LIN {X 0,Y 291.883,Z 681.921,A -85,B 0,C 180,E1 -16741.379,E2 -16741.379} C_VEL
LIN {X 0,Y 291.735,Z 681.939,A -85,B 0,C 180,E1 -16746.918,E2 -16746.918} C_VEL
LIN {X 0,Y 291.622,Z 681.967,A -85,B 0,C 180,E1 -16749.712,E2 -16749.712} C_VEL
LIN {X 0,Y 291.513,Z 681.968,A -85,B 0,C 180,E1 -16753.95,E2 -16753.95} C_VEL
LIN {X 0,Y 291.479,Z 681.972,A -85,B 0,C 180,E1 -16756.818,E2 -16756.818} C_VEL
LIN {X 0,Y 291.477,Z 681.99,A -85,B 0,C 180,E1 -16759.893,E2 -16759.893} C_VEL
LIN {X 0,Y 291.416,Z 681.996,A -85,B 0,C 180,E1 -16764.203,E2 -16764.203} C_VEL
LIN {X 0,Y 291.414,Z 681.938,A -85,B 0,C 180,E1 -16767.272,E2 -16767.272} C_VEL
LIN {X 0,Y 291.329,Z 681.954,A -85,B 0,C 180,E1 -16770.437,E2 -16770.437} C_VEL
LIN {X 0,Y 291.337,Z 681.982,A -85,B 0,C 180,E1 -16773.699,E2 -16773.699} C_VEL
LIN {X 0,Y 291.422,Z 682.063,A -85,B 0,C 180,E1 -16777.556,E2 -16777.556} C_VEL
LIN {X 0,Y 291.562,Z 682.874,A -85,B 0,C 180,E1 -16777.957,E2 -16777.957} C_VEL
LIN {X 0,Y 292.964,Z 685.685,A -85,B 0,C 180,E1 -16778.482,E2 -16778.482} C_VEL
LIN {X 0,Y 295.139,Z 687.721,A -85,B 0,C 180,E1 -16779.091,E2 -16779.091} C_VEL
LIN {X 0,Y 297.372,Z 691.036,A -85,B 0,C 180,E1 -16779.745,E2 -16779.745} C_VEL
LIN {X 0,Y 299.349,Z 693.065,A -85,B 0,C 180,E1 -16780.308,E2 -16780.308} C_VEL
LIN {X 0,Y 302.176,Z 696.689,A -85,B 0,C 180,E1 -16781.129,E2 -16781.129} C_VEL
LIN {X 0,Y 304.398,Z 698.863,A -85,B 0,C 180,E1 -16781.754,E2 -16781.754} C_VEL
LIN {X 0,Y 307.399,Z 702.53,A -85,B 0,C 180,E1 -16782.702,E2 -16782.702} C_VEL
LIN {X 0,Y 309.651,Z 704.604,A -85,B 0,C 180,E1 -16783.366,E2 -16783.366} C_VEL
LIN {X 0,Y 312.93,Z 708.385,A -85,B 0,C 180,E1 -16784.462,E2 -16784.462} C_VEL
LIN {X 0,Y 315.506,Z 710.671,A -85,B 0,C 180,E1 -16785.293,E2 -16785.293} C_VEL
LIN {X 0,Y 318.764,Z 714.434,A -85,B 0,C 180,E1 -16786.475,E2 -16786.475} C_VEL
LIN {X 0,Y 321.428,Z 716.849,A -85,B 0,C 180,E1 -16787.424,E2 -16787.424} C_VEL
LIN {X 0,Y 324.974,Z 720.767,A -85,B 0,C 180,E1 -16788.792,E2 -16788.792} C_VEL
LIN {X 0,Y 327.213,Z 722.862,A -85,B 0,C 180,E1 -16789.66,E2 -16789.66} C_VEL
LIN {X 0,Y 330.789,Z 726.747,A -85,B 0,C 180,E1 -16791.088,E2 -16791.088} C_VEL
LIN {X 0,Y 333.202,Z 728.975,A -85,B 0,C 180,E1 -16792.056,E2 -16792.056} C_VEL
LIN {X 0,Y 336.504,Z 732.572,A -85,B 0,C 180,E1 -16793.429,E2 -16793.429} C_VEL
LIN {X 0,Y 339.383,Z 735.138,A -85,B 0,C 180,E1 -16794.624,E2 -16794.624} C_VEL
LIN {X 0,Y 343.284,Z 739.204,A -85,B 0,C 180,E1 -16796.335,E2 -16796.335} C_VEL
LIN {X 0,Y 346.175,Z 741.646,A -85,B 0,C 180,E1 -16797.613,E2 -16797.613} C_VEL
LIN {X 0,Y 349.884,Z 745.493,A -85,B 0,C 180,E1 -16799.349,E2 -16799.349} C_VEL
LIN {X 0,Y 352.817,Z 747.883,A -85,B 0,C 180,E1 -16800.742,E2 -16800.742} C_VEL
LIN {X 0,Y 356.182,Z 751.516,A -85,B 0,C 180,E1 -16802.455,E2 -16802.455} C_VEL
LIN {X 0,Y 359.846,Z 754.425,A -85,B 0,C 180,E1 -16804.388,E2 -16804.388} C_VEL
LIN {X 0,Y 363.148,Z 758.001,A -85,B 0,C 180,E1 -16806.288,E2 -16806.288} C_VEL
LIN {X 0,Y 366.688,Z 760.486,A -85,B 0,C 180,E1 -16808.414,E2 -16808.414} C_VEL
LIN {X 0,Y 367.985,Z 761.786,A -85,B 0,C 180,E1 -16809.246,E2 -16809.246} C_VEL
LIN {X 0,Y 370.733,Z 764.739,A -85,B 0,C 180,E1 -16811.2,E2 -16811.2} C_VEL
LIN {X 0,Y 373.538,Z 766.766,A -85,B 0,C 180,E1 -16813.28,E2 -16813.28} C_VEL
LIN {X 0,Y 375.474,Z 767.943,A -85,B 0,C 180,E1 -16814.874,E2 -16814.874} C_VEL
LIN {X 0,Y 377.522,Z 770.55,A -85,B 0,C 180,E1 -16816.885,E2 -16816.885} C_VEL
LIN {X 0,Y 379.42,Z 772.303,A -85,B 0,C 180,E1 -16819.024,E2 -16819.024} C_VEL
LIN {X 0,Y 381.332,Z 773.414,A -85,B 0,C 180,E1 -16821.522,E2 -16821.522} C_VEL
LIN {X 0,Y 382.798,Z 774.146,A -85,B 0,C 180,E1 -16824.133,E2 -16824.133} C_VEL
LIN {X 0,Y 383.462,Z 774.602,A -85,B 0,C 180,E1 -16825.796,E2 -16825.796} C_VEL
LIN {X 0,Y 384.005,Z 774.796,A -85,B 0,C 180,E1 -16827.902,E2 -16827.902} C_VEL
LIN {X 0,Y 384.204,Z 774.867,A -85,B 0,C 180,E1 -16830,E2 -16830} C_VEL
LIN {X 0,Y 384.005,Z 774.797,A -85,B 0,C 180,E1 -16832.098,E2 -16832.098} C_VEL
LIN {X 0,Y 383.313,Z 774.45,A -85,B 0,C 180,E1 -16834.646,E2 -16834.646} C_VEL
LIN {X 0,Y 382.015,Z 773.719,A -85,B 0,C 180,E1 -16837.399,E2 -16837.399} C_VEL
LIN {X 0,Y 380.152,Z 772.82,A -85,B 0,C 180,E1 -16840.106,E2 -16840.106} C_VEL
LIN {X 0,Y 378.053,Z 771.142,A -85,B 0,C 180,E1 -16842.519,E2 -16842.519} C_VEL
LIN {X 0,Y 375.891,Z 768.596,A -85,B 0,C 180,E1 -16844.721,E2 -16844.721} C_VEL
LIN {X 0,Y 374.994,Z 767.485,A -85,B 0,C 180,E1 -16845.55,E2 -16845.55} C_VEL
LIN {X 0,Y 371.895,Z 765.67,A -85,B 0,C 180,E1 -16847.968,E2 -16847.968} C_VEL
LIN {X 0,Y 368.875,Z 762.885,A -85,B 0,C 180,E1 -16850.115,E2 -16850.115} C_VEL
LIN {X 0,Y 366.9,Z 760.575,A -85,B 0,C 180,E1 -16851.458,E2 -16851.458} C_VEL
LIN {X 0,Y 363.407,Z 758.198,A -85,B 0,C 180,E1 -16853.568,E2 -16853.568} C_VEL
LIN {X 0,Y 359.968,Z 754.568,A -85,B 0,C 180,E1 -16855.543,E2 -16855.543} C_VEL
LIN {X 0,Y 357.887,Z 752.872,A -85,B 0,C 180,E1 -16856.654,E2 -16856.654} C_VEL
LIN {X 0,Y 354.468,Z 749.835,A -85,B 0,C 180,E1 -16858.414,E2 -16858.414} C_VEL
LIN {X 0,Y 351.836,Z 746.961,A -85,B 0,C 180,E1 -16859.736,E2 -16859.736} C_VEL
LIN {X 0,Y 347.935,Z 743.618,A -85,B 0,C 180,E1 -16861.578,E2 -16861.578} C_VEL
LIN {X 0,Y 344.914,Z 740.41,A -85,B 0,C 180,E1 -16862.971,E2 -16862.971} C_VEL
LIN {X 0,Y 341.103,Z 737.112,A -85,B 0,C 180,E1 -16864.623,E2 -16864.623} C_VEL
LIN {X 0,Y 338.238,Z 733.951,A -85,B 0,C 180,E1 -16865.871,E2 -16865.871} C_VEL
LIN {X 0,Y 334.572,Z 730.578,A -85,B 0,C 180,E1 -16867.379,E2 -16867.379} C_VEL
LIN {X 0,Y 332.005,Z 727.717,A -85,B 0,C 180,E1 -16868.444,E2 -16868.444} C_VEL
LIN {X 0,Y 328.279,Z 724.166,A -85,B 0,C 180,E1 -16869.919,E2 -16869.919} C_VEL
LIN {X 0,Y 326.08,Z 721.692,A -85,B 0,C 180,E1 -16870.78,E2 -16870.78} C_VEL
LIN {X 0,Y 322.545,Z 718.298,A -85,B 0,C 180,E1 -16872.134,E2 -16872.134} C_VEL
LIN {X 0,Y 320.523,Z 715.855,A -85,B 0,C 180,E1 -16872.919,E2 -16872.919} C_VEL
LIN {X 0,Y 316.761,Z 712.285,A -85,B 0,C 180,E1 -16874.256,E2 -16874.256} C_VEL
LIN {X 0,Y 314.552,Z 709.736,A -85,B 0,C 180,E1 -16875.024,E2 -16875.024} C_VEL
LIN {X 0,Y 310.731,Z 706.058,A -85,B 0,C 180,E1 -16876.271,E2 -16876.271} C_VEL
LIN {X 0,Y 308.685,Z 703.611,A -85,B 0,C 180,E1 -16876.92,E2 -16876.92} C_VEL
LIN {X 0,Y 305.31,Z 700.201,A -85,B 0,C 180,E1 -16877.943,E2 -16877.943} C_VEL
LIN {X 0,Y 303.441,Z 697.755,A -85,B 0,C 180,E1 -16878.528,E2 -16878.528} C_VEL
LIN {X 0,Y 300.227,Z 694.445,A -85,B 0,C 180,E1 -16879.424,E2 -16879.424} C_VEL
LIN {X 0,Y 298.66,Z 692.237,A -85,B 0,C 180,E1 -16879.895,E2 -16879.895} C_VEL
LIN {X 0,Y 296.057,Z 689.359,A -85,B 0,C 180,E1 -16880.628,E2 -16880.628} C_VEL
LIN {X 0,Y 294.621,Z 687.154,A -85,B 0,C 180,E1 -16881.056,E2 -16881.056} C_VEL
LIN {X 0,Y 292.502,Z 685.027,A -85,B 0,C 180,E1 -16881.659,E2 -16881.659} C_VEL
LIN {X 0,Y 291.49,Z 682.559,A -85,B 0,C 180,E1 -16882.138,E2 -16882.138} C_VEL
LIN {X 0,Y 291.422,Z 682.053,A -85,B 0,C 180,E1 -16882.444,E2 -16882.444} C_VEL
LIN {X 0,Y 291.337,Z 681.982,A -85,B 0,C 180,E1 -16886.301,E2 -16886.301} C_VEL
LIN {X 0,Y 291.379,Z 681.937,A -85,B 0,C 180,E1 -16890.26,E2 -16890.26} C_VEL
LIN {X 0,Y 291.408,Z 681.977,A -85,B 0,C 180,E1 -16894.272,E2 -16894.272} C_VEL
LIN {X 0,Y 291.384,Z 681.984,A -85,B 0,C 180,E1 -16897.3,E2 -16897.3} C_VEL
LIN {X 0,Y 291.497,Z 681.986,A -85,B 0,C 180,E1 -16900.273,E2 -16900.273} C_VEL
LIN {X 0,Y 291.533,Z 681.981,A -85,B 0,C 180,E1 -16904.635,E2 -16904.635} C_VEL
LIN {X 0,Y 291.529,Z 681.973,A -85,B 0,C 180,E1 -16908.881,E2 -16908.881} C_VEL
LIN {X 0,Y 291.694,Z 681.939,A -85,B 0,C 180,E1 -16911.689,E2 -16911.689} C_VEL
LIN {X 0,Y 291.624,Z 681.969,A -85,B 0,C 180,E1 -16914.469,E2 -16914.469} C_VEL
LIN {X 0,Y 291.883,Z 681.922,A -85,B 0,C 180,E1 -16918.621,E2 -16918.621} C_VEL
LIN {X 0,Y 291.883,Z 681.927,A -85,B 0,C 180,E1 -16921.38,E2 -16921.38} C_VEL
LIN {X 0,Y 291.736,Z 681.937,A -85,B 0,C 180,E1 -16926.918,E2 -16926.918} C_VEL
LIN {X 0,Y 291.623,Z 681.961,A -85,B 0,C 180,E1 -16929.712,E2 -16929.712} C_VEL
LIN {X 0,Y 291.511,Z 681.966,A -85,B 0,C 180,E1 -16933.877,E2 -16933.877} C_VEL
LIN {X 0,Y 290.876,Z 682.062,A -85,B 0,C 180,E1 -16935.03,E2 -16935.03} C_VEL
LIN {X 0,Y 287.969,Z 682.41,A -85,B 0,C 180,E1 -16936.904,E2 -16936.904} C_VEL
LIN {X 0,Y 285.489,Z 682.717,A -85,B 0,C 180,E1 -16938.427,E2 -16938.427} C_VEL
LIN {X 0,Y 284.448,Z 682.86,A -85,B 0,C 180,E1 -16939.608,E2 -16939.608} C_VEL
LIN {X 0,Y 284.378,Z 682.873,A -85,B 0,C 180,E1 -16940.009,E2 -16940.009} C_VEL
LIN {X 0,Y 284.363,Z 682.867,A -85,B 0,C 180,E1 -16943.876,E2 -16943.876} C_VEL
LIN {X 0,Y 284.391,Z 682.814,A -85,B 0,C 180,E1 -16947.174,E2 -16947.174} C_VEL
LIN {X 0,Y 284.29,Z 682.846,A -85,B 0,C 180,E1 -16951.275,E2 -16951.275} C_VEL
LIN {X 0,Y 284.378,Z 683.065,A -85,B 0,C 180,E1 -16954.785,E2 -16954.785} C_VEL
LIN {X 0,Y 285.219,Z 685.498,A -85,B 0,C 180,E1 -16955.965,E2 -16955.965} C_VEL
LIN {X 0,Y 288.149,Z 690.097,A -85,B 0,C 180,E1 -16957.023,E2 -16957.023} C_VEL
LIN {X 0,Y 290.383,Z 693.289,A -85,B 0,C 180,E1 -16957.725,E2 -16957.725} C_VEL
LIN {X 0,Y 294.154,Z 698.909,A -85,B 0,C 180,E1 -16958.872,E2 -16958.872} C_VEL
LIN {X 0,Y 298.001,Z 704.821,A -85,B 0,C 180,E1 -16959.991,E2 -16959.991} C_VEL
LIN {X 0,Y 303.606,Z 713.81,A -85,B 0,C 180,E1 -16961.541,E2 -16961.541} C_VEL
LIN {X 0,Y 311.488,Z 727.717,A -85,B 0,C 180,E1 -16963.596,E2 -16963.596} C_VEL
LIN {X 0,Y 319,Z 742.269,A -85,B 0,C 180,E1 -16965.437,E2 -16965.437} C_VEL
LIN {X 0,Y 326.807,Z 759.311,A -85,B 0,C 180,E1 -16967.26,E2 -16967.26} C_VEL
LIN {X 0,Y 326.66,Z 767.163,A -85,B 0,C 180,E1 -16967.465,E2 -16967.465} C_VEL
LIN {X 0,Y 320.836,Z 891.245,A -85,B 0,C 180,E1 -16970.192,E2 -16970.192} C_VEL
LIN {X 0,Y 319.83,Z 903.367,A -85,B 0,C 180,E1 -16970.567,E2 -16970.567} C_VEL
LIN {X 0,Y 318.218,Z 916.468,A -85,B 0,C 180,E1 -16971.094,E2 -16971.094} C_VEL
LIN {X 0,Y 316.345,Z 928.835,A -85,B 0,C 180,E1 -16971.738,E2 -16971.738} C_VEL
LIN {X 0,Y 314.451,Z 940.221,A -85,B 0,C 180,E1 -16972.481,E2 -16972.481} C_VEL
LIN {X 0,Y 311.776,Z 953.453,A -85,B 0,C 180,E1 -16973.521,E2 -16973.521} C_VEL
LIN {X 0,Y 308.946,Z 966.189,A -85,B 0,C 180,E1 -16974.745,E2 -16974.745} C_VEL
LIN {X 0,Y 306.236,Z 977.219,A -85,B 0,C 180,E1 -16975.992,E2 -16975.992} C_VEL
LIN {X 0,Y 303.306,Z 987.98,A -85,B 0,C 180,E1 -16977.404,E2 -16977.404} C_VEL
LIN {X 0,Y 300.348,Z 998.478,A -85,B 0,C 180,E1 -16979.018,E2 -16979.018} C_VEL
LIN {X 0,Y 297.156,Z 1009.247,A -85,B 0,C 180,E1 -16980.959,E2 -16980.959} C_VEL
LIN {X 0,Y 294.2,Z 1018.944,A -85,B 0,C 180,E1 -16983.008,E2 -16983.008} C_VEL
LIN {X 0,Y 291.622,Z 1027.282,A -85,B 0,C 180,E1 -16985.056,E2 -16985.056} C_VEL
LIN {X 0,Y 289.416,Z 1034.604,A -85,B 0,C 180,E1 -16987.137,E2 -16987.137} C_VEL
LIN {X 0,Y 287.576,Z 1041.038,A -85,B 0,C 180,E1 -16989.246,E2 -16989.246} C_VEL
LIN {X 0,Y 285.518,Z 1048.301,A -85,B 0,C 180,E1 -16992.081,E2 -16992.081} C_VEL
LIN {X 0,Y 284.217,Z 1053.771,A -85,B 0,C 180,E1 -16994.66,E2 -16994.66} C_VEL
LIN {X 0,Y 283.364,Z 1058.06,A -85,B 0,C 180,E1 -16997.102,E2 -16997.102} C_VEL
LIN {X 0,Y 282.649,Z 1062.062,A -85,B 0,C 180,E1 -16999.977,E2 -16999.977} C_VEL
LIN {X 0,Y 282.491,Z 1063.74,A -85,B 0,C 180,E1 -17001.416,E2 -17001.416} C_VEL
LIN {X 0,Y 282.327,Z 1066.473,A -85,B 0,C 180,E1 -17004.699,E2 -17004.699} C_VEL
LIN {X 0,Y 282.322,Z 1067.686,A -85,B 0,C 180,E1 -17007.146,E2 -17007.146} C_VEL
LIN {X 0,Y 282.354,Z 1068.174,A -85,B 0,C 180,E1 -17010,E2 -17010} C_VEL
LIN {X 0,Y 282.322,Z 1067.686,A -85,B 0,C 180,E1 -17012.854,E2 -17012.854} C_VEL
LIN {X 0,Y 282.337,Z 1066.213,A -85,B 0,C 180,E1 -17015.714,E2 -17015.714} C_VEL
LIN {X 0,Y 282.491,Z 1063.74,A -85,B 0,C 180,E1 -17018.584,E2 -17018.584} C_VEL
LIN {X 0,Y 283.143,Z 1059.149,A -85,B 0,C 180,E1 -17022.18,E2 -17022.18} C_VEL
LIN {X 0,Y 283.857,Z 1055.657,A -85,B 0,C 180,E1 -17024.335,E2 -17024.335} C_VEL
LIN {X 0,Y 285.113,Z 1049.924,A -85,B 0,C 180,E1 -17027.205,E2 -17027.205} C_VEL
LIN {X 0,Y 286.481,Z 1044.862,A -85,B 0,C 180,E1 -17029.34,E2 -17029.34} C_VEL
LIN {X 0,Y 288.614,Z 1037.389,A -85,B 0,C 180,E1 -17031.985,E2 -17031.985} C_VEL
LIN {X 0,Y 290.838,Z 1029.842,A -85,B 0,C 180,E1 -17034.254,E2 -17034.254} C_VEL
LIN {X 0,Y 293.279,Z 1021.874,A -85,B 0,C 180,E1 -17036.315,E2 -17036.315} C_VEL
LIN {X 0,Y 296.095,Z 1012.762,A -85,B 0,C 180,E1 -17038.34,E2 -17038.34} C_VEL
LIN {X 0,Y 298.653,Z 1004.194,A -85,B 0,C 180,E1 -17040.003,E2 -17040.003} C_VEL
LIN {X 0,Y 302.032,Z 992.329,A -85,B 0,C 180,E1 -17041.962,E2 -17041.962} C_VEL
LIN {X 0,Y 304.877,Z 982.168,A -85,B 0,C 180,E1 -17043.391,E2 -17043.391} C_VEL
LIN {X 0,Y 307.895,Z 970.502,A -85,B 0,C 180,E1 -17044.794,E2 -17044.794} C_VEL
LIN {X 0,Y 310.683,Z 958.479,A -85,B 0,C 180,E1 -17046.025,E2 -17046.025} C_VEL
LIN {X 0,Y 313.301,Z 946.163,A -85,B 0,C 180,E1 -17047.074,E2 -17047.074} C_VEL
LIN {X 0,Y 315.554,Z 933.62,A -85,B 0,C 180,E1 -17047.97,E2 -17047.97} C_VEL
LIN {X 0,Y 317.658,Z 920.196,A -85,B 0,C 180,E1 -17048.733,E2 -17048.733} C_VEL
LIN {X 0,Y 319.381,Z 907.283,A -85,B 0,C 180,E1 -17049.295,E2 -17049.295} C_VEL
LIN {X 0,Y 320.724,Z 893.792,A -85,B 0,C 180,E1 -17049.732,E2 -17049.732} C_VEL
LIN {X 0,Y 322.084,Z 865.058,A -85,B 0,C 180,E1 -17050.419,E2 -17050.419} C_VEL
LIN {X 0,Y 326.923,Z 759.58,A -85,B 0,C 180,E1 -17052.714,E2 -17052.714} C_VEL
LIN {X 0,Y 320.449,Z 745.364,A -85,B 0,C 180,E1 -17054.216,E2 -17054.216} C_VEL
LIN {X 0,Y 313.198,Z 730.801,A -85,B 0,C 180,E1 -17055.979,E2 -17055.979} C_VEL
LIN {X 0,Y 305.161,Z 716.52,A -85,B 0,C 180,E1 -17058.04,E2 -17058.04} C_VEL
LIN {X 0,Y 299.247,Z 706.697,A -85,B 0,C 180,E1 -17059.66,E2 -17059.66} C_VEL
LIN {X 0,Y 295.583,Z 701.084,A -85,B 0,C 180,E1 -17060.707,E2 -17060.707} C_VEL
LIN {X 0,Y 292.286,Z 696.088,A -85,B 0,C 180,E1 -17061.69,E2 -17061.69} C_VEL
LIN {X 0,Y 288.27,Z 690.224,A -85,B 0,C 180,E1 -17062.941,E2 -17062.941} C_VEL
LIN {X 0,Y 285.408,Z 685.904,A -85,B 0,C 180,E1 -17063.918,E2 -17063.918} C_VEL
LIN {X 0,Y 284.43,Z 683.299,A -85,B 0,C 180,E1 -17065.077,E2 -17065.077} C_VEL
LIN {X 0,Y 284.307,Z 682.849,A -85,B 0,C 180,E1 -17065.78,E2 -17065.78} C_VEL
LIN {X 0,Y 284.353,Z 682.808,A -85,B 0,C 180,E1 -17070.375,E2 -17070.375} C_VEL
LIN {X 0,Y 284.371,Z 682.832,A -85,B 0,C 180,E1 -17073.586,E2 -17073.586} C_VEL
LIN {X 0,Y 284.36,Z 682.86,A -85,B 0,C 180,E1 -17076.706,E2 -17076.706} C_VEL
LIN {X 0,Y 284.399,Z 682.855,A -85,B 0,C 180,E1 -17081.261,E2 -17081.261} C_VEL
LIN {X 0,Y 284.472,Z 682.864,A -85,B 0,C 180,E1 -17084.469,E2 -17084.469} C_VEL
LIN {X 0,Y 284.483,Z 682.851,A -85,B 0,C 180,E1 -17088.601,E2 -17088.601} C_VEL
LIN {X 0,Y 284.65,Z 682.815,A -85,B 0,C 180,E1 -17091.481,E2 -17091.481} C_VEL
LIN {X 0,Y 284.595,Z 682.844,A -85,B 0,C 180,E1 -17094.331,E2 -17094.331} C_VEL
LIN {X 0,Y 284.849,Z 682.8,A -85,B 0,C 180,E1 -17098.586,E2 -17098.586} C_VEL
LIN {X 0,Y 284.849,Z 682.796,A -85,B 0,C 180,E1 -17101.413,E2 -17101.413} C_VEL
LIN {X 0,Y 284.687,Z 682.815,A -85,B 0,C 180,E1 -17107.09,E2 -17107.09} C_VEL
LIN {X 0,Y 284.559,Z 682.85,A -85,B 0,C 180,E1 -17109.955,E2 -17109.955} C_VEL
LIN {X 0,Y 284.47,Z 682.849,A -85,B 0,C 180,E1 -17114.303,E2 -17114.303} C_VEL
LIN {X 0,Y 284.419,Z 682.848,A -85,B 0,C 180,E1 -17117.248,E2 -17117.248} C_VEL
LIN {X 0,Y 284.412,Z 682.87,A -85,B 0,C 180,E1 -17120.239,E2 -17120.239} C_VEL
LIN {X 0,Y 284.378,Z 682.868,A -85,B 0,C 180,E1 -17123.882,E2 -17123.882} C_VEL
LIN {X 0,Y 284.389,Z 682.813,A -85,B 0,C 180,E1 -17127.173,E2 -17127.173} C_VEL
LIN {X 0,Y 284.288,Z 682.848,A -85,B 0,C 180,E1 -17131.274,E2 -17131.274} C_VEL
LIN {X 0,Y 284.335,Z 682.975,A -85,B 0,C 180,E1 -17135.726,E2 -17135.726} C_VEL
LIN {X 0,Y 284.593,Z 684.124,A -85,B 0,C 180,E1 -17136.2,E2 -17136.2} C_VEL
LIN {X 0,Y 286.249,Z 686.848,A -85,B 0,C 180,E1 -17136.793,E2 -17136.793} C_VEL
LIN {X 0,Y 288.169,Z 688.504,A -85,B 0,C 180,E1 -17137.371,E2 -17137.371} C_VEL
LIN {X 0,Y 290.198,Z 691.815,A -85,B 0,C 180,E1 -17138.027,E2 -17138.027} C_VEL
LIN {X 0,Y 292.166,Z 693.903,A -85,B 0,C 180,E1 -17138.602,E2 -17138.602} C_VEL
LIN {X 0,Y 294.925,Z 697.535,A -85,B 0,C 180,E1 -17139.411,E2 -17139.411} C_VEL
LIN {X 0,Y 296.587,Z 699.355,A -85,B 0,C 180,E1 -17139.871,E2 -17139.871} C_VEL
LIN {X 0,Y 299.727,Z 703.115,A -85,B 0,C 180,E1 -17140.782,E2 -17140.782} C_VEL
LIN {X 0,Y 301.55,Z 704.967,A -85,B 0,C 180,E1 -17141.288,E2 -17141.288} C_VEL
LIN {X 0,Y 304.924,Z 708.829,A -85,B 0,C 180,E1 -17142.301,E2 -17142.301} C_VEL
LIN {X 0,Y 307.205,Z 711.064,A -85,B 0,C 180,E1 -17142.989,E2 -17142.989} C_VEL
LIN {X 0,Y 310.726,Z 714.847,A -85,B 0,C 180,E1 -17144.099,E2 -17144.099} C_VEL
LIN {X 0,Y 313.289,Z 717.232,A -85,B 0,C 180,E1 -17144.932,E2 -17144.932} C_VEL
LIN {X 0,Y 316.936,Z 721.117,A -85,B 0,C 180,E1 -17146.198,E2 -17146.198} C_VEL
LIN {X 0,Y 319.534,Z 723.555,A -85,B 0,C 180,E1 -17147.114,E2 -17147.114} C_VEL
LIN {X 0,Y 323.35,Z 727.582,A -85,B 0,C 180,E1 -17148.563,E2 -17148.563} C_VEL
LIN {X 0,Y 325.397,Z 729.609,A -85,B 0,C 180,E1 -17149.36,E2 -17149.36} C_VEL
LIN {X 0,Y 329.352,Z 733.702,A -85,B 0,C 180,E1 -17150.921,E2 -17150.921} C_VEL
LIN {X 0,Y 331.476,Z 735.7,A -85,B 0,C 180,E1 -17151.759,E2 -17151.759} C_VEL
LIN {X 0,Y 335.122,Z 739.522,A -85,B 0,C 180,E1 -17153.263,E2 -17153.263} C_VEL
LIN {X 0,Y 337.594,Z 741.712,A -85,B 0,C 180,E1 -17154.281,E2 -17154.281} C_VEL
LIN {X 0,Y 341.824,Z 746.022,A -85,B 0,C 180,E1 -17156.117,E2 -17156.117} C_VEL
LIN {X 0,Y 344.393,Z 748.122,A -85,B 0,C 180,E1 -17157.232,E2 -17157.232} C_VEL
LIN {X 0,Y 348.497,Z 752.348,A -85,B 0,C 180,E1 -17159.148,E2 -17159.148} C_VEL
LIN {X 0,Y 351.328,Z 754.663,A -85,B 0,C 180,E1 -17160.483,E2 -17160.483} C_VEL
LIN {X 0,Y 354.774,Z 758.317,A -85,B 0,C 180,E1 -17162.223,E2 -17162.223} C_VEL
LIN {X 0,Y 358.497,Z 761.249,A -85,B 0,C 180,E1 -17164.156,E2 -17164.156} C_VEL
LIN {X 0,Y 361.813,Z 764.816,A -85,B 0,C 180,E1 -17166.056,E2 -17166.056} C_VEL
LIN {X 0,Y 365.46,Z 767.374,A -85,B 0,C 180,E1 -17168.209,E2 -17168.209} C_VEL
LIN {X 0,Y 366.985,Z 768.904,A -85,B 0,C 180,E1 -17169.187,E2 -17169.187} C_VEL
LIN {X 0,Y 369.762,Z 771.808,A -85,B 0,C 180,E1 -17171.149,E2 -17171.149} C_VEL
LIN {X 0,Y 372.798,Z 773.899,A -85,B 0,C 180,E1 -17173.392,E2 -17173.392} C_VEL
LIN {X 0,Y 374.467,Z 774.989,A -85,B 0,C 180,E1 -17174.767,E2 -17174.767} C_VEL
LIN {X 0,Y 376.711,Z 777.756,A -85,B 0,C 180,E1 -17176.96,E2 -17176.96} C_VEL
LIN {X 0,Y 378.895,Z 779.644,A -85,B 0,C 180,E1 -17179.442,E2 -17179.442} C_VEL
LIN {X 0,Y 380.888,Z 780.66,A -85,B 0,C 180,E1 -17182.17,E2 -17182.17} C_VEL
LIN {X 0,Y 382.222,Z 781.318,A -85,B 0,C 180,E1 -17184.725,E2 -17184.725} C_VEL
LIN {X 0,Y 382.92,Z 781.719,A -85,B 0,C 180,E1 -17186.844,E2 -17186.844} C_VEL
LIN {X 0,Y 383.256,Z 781.952,A -85,B 0,C 180,E1 -17188.949,E2 -17188.949} C_VEL
LIN {X 0,Y 383.256,Z 781.954,A -85,B 0,C 180,E1 -17191.051,E2 -17191.051} C_VEL
LIN {X 0,Y 382.92,Z 781.72,A -85,B 0,C 180,E1 -17193.156,E2 -17193.156} C_VEL
LIN {X 0,Y 382.221,Z 781.319,A -85,B 0,C 180,E1 -17195.275,E2 -17195.275} C_VEL
LIN {X 0,Y 380.716,Z 780.603,A -85,B 0,C 180,E1 -17198.102,E2 -17198.102} C_VEL
LIN {X 0,Y 378.681,Z 779.508,A -85,B 0,C 180,E1 -17200.812,E2 -17200.812} C_VEL
LIN {X 0,Y 376.398,Z 777.432,A -85,B 0,C 180,E1 -17203.341,E2 -17203.341} C_VEL
LIN {X 0,Y 373.87,Z 774.397,A -85,B 0,C 180,E1 -17205.753,E2 -17205.753} C_VEL
LIN {X 0,Y 370.944,Z 772.712,A -85,B 0,C 180,E1 -17208.016,E2 -17208.016} C_VEL
LIN {X 0,Y 367.882,Z 769.987,A -85,B 0,C 180,E1 -17210.171,E2 -17210.171} C_VEL
LIN {X 0,Y 365.689,Z 767.495,A -85,B 0,C 180,E1 -17211.649,E2 -17211.649} C_VEL
LIN {X 0,Y 361.814,Z 764.813,A -85,B 0,C 180,E1 -17213.944,E2 -17213.944} C_VEL
LIN {X 0,Y 358.266,Z 760.959,A -85,B 0,C 180,E1 -17215.978,E2 -17215.978} C_VEL
LIN {X 0,Y 354.117,Z 757.698,A -85,B 0,C 180,E1 -17218.107,E2 -17218.107} C_VEL
LIN {X 0,Y 350.483,Z 753.825,A -85,B 0,C 180,E1 -17219.935,E2 -17219.935} C_VEL
LIN {X 0,Y 346.319,Z 750.308,A -85,B 0,C 180,E1 -17221.866,E2 -17221.866} C_VEL
LIN {X 0,Y 343.393,Z 747.213,A -85,B 0,C 180,E1 -17223.207,E2 -17223.207} C_VEL
LIN {X 0,Y 339.347,Z 743.711,A -85,B 0,C 180,E1 -17224.95,E2 -17224.95} C_VEL
LIN {X 0,Y 336.351,Z 740.496,A -85,B 0,C 180,E1 -17226.233,E2 -17226.233} C_VEL
LIN {X 0,Y 332.438,Z 736.874,A -85,B 0,C 180,E1 -17227.833,E2 -17227.833} C_VEL
LIN {X 0,Y 329.919,Z 734.125,A -85,B 0,C 180,E1 -17228.863,E2 -17228.863} C_VEL
LIN {X 0,Y 326.086,Z 730.417,A -85,B 0,C 180,E1 -17230.368,E2 -17230.368} C_VEL
LIN {X 0,Y 323.933,Z 728.077,A -85,B 0,C 180,E1 -17231.218,E2 -17231.218} C_VEL
LIN {X 0,Y 320.136,Z 724.307,A -85,B 0,C 180,E1 -17232.658,E2 -17232.658} C_VEL
LIN {X 0,Y 318.08,Z 722.093,A -85,B 0,C 180,E1 -17233.396,E2 -17233.396} C_VEL
LIN {X 0,Y 314.332,Z 718.464,A -85,B 0,C 180,E1 -17234.718,E2 -17234.718} C_VEL
LIN {X 0,Y 312.096,Z 715.979,A -85,B 0,C 180,E1 -17235.458,E2 -17235.458} C_VEL
LIN {X 0,Y 308.241,Z 712.32,A -85,B 0,C 180,E1 -17236.693,E2 -17236.693} C_VEL
LIN {X 0,Y 305.684,Z 709.496,A -85,B 0,C 180,E1 -17237.467,E2 -17237.467} C_VEL
LIN {X 0,Y 302.279,Z 705.9,A -85,B 0,C 180,E1 -17238.5,E2 -17238.5} C_VEL
LIN {X 0,Y 300.159,Z 703.487,A -85,B 0,C 180,E1 -17239.099,E2 -17239.099} C_VEL
LIN {X 0,Y 296.792,Z 699.704,A -85,B 0,C 180,E1 -17240.067,E2 -17240.067} C_VEL
LIN {X 0,Y 295.323,Z 697.904,A -85,B 0,C 180,E1 -17240.48,E2 -17240.48} C_VEL
LIN {X 0,Y 292.475,Z 694.397,A -85,B 0,C 180,E1 -17241.302,E2 -17241.302} C_VEL
LIN {X 0,Y 291.184,Z 692.8,A -85,B 0,C 180,E1 -17241.685,E2 -17241.685} C_VEL
LIN {X 0,Y 288.743,Z 689.711,A -85,B 0,C 180,E1 -17242.431,E2 -17242.431} C_VEL
LIN {X 0,Y 287.737,Z 688.062,A -85,B 0,C 180,E1 -17242.761,E2 -17242.761} C_VEL
LIN {X 0,Y 285.433,Z 685.847,A -85,B 0,C 180,E1 -17243.47,E2 -17243.47} C_VEL
LIN {X 0,Y 284.446,Z 683.591,A -85,B 0,C 180,E1 -17243.925,E2 -17243.925} C_VEL
LIN {X 0,Y 284.311,Z 682.895,A -85,B 0,C 180,E1 -17244.343,E2 -17244.343} C_VEL
LIN {X 0,Y 284.288,Z 682.848,A -85,B 0,C 180,E1 -17248.726,E2 -17248.726} C_VEL
LIN {X 0,Y 284.389,Z 682.813,A -85,B 0,C 180,E1 -17252.827,E2 -17252.827} C_VEL
LIN {X 0,Y 284.368,Z 682.861,A -85,B 0,C 180,E1 -17256.708,E2 -17256.708} C_VEL
LIN {X 0,Y 284.424,Z 682.87,A -85,B 0,C 180,E1 -17259.874,E2 -17259.874} C_VEL
LIN {X 0,Y 284.471,Z 682.861,A -85,B 0,C 180,E1 -17264.47,E2 -17264.47} C_VEL
LIN {X 0,Y 284.48,Z 682.845,A -85,B 0,C 180,E1 -17268.602,E2 -17268.602} C_VEL
LIN {X 0,Y 284.646,Z 682.818,A -85,B 0,C 180,E1 -17271.481,E2 -17271.481} C_VEL
LIN {X 0,Y 284.594,Z 682.843,A -85,B 0,C 180,E1 -17274.332,E2 -17274.332} C_VEL
LIN {X 0,Y 284.849,Z 682.797,A -85,B 0,C 180,E1 -17278.587,E2 -17278.587} C_VEL
LIN {X 0,Y 284.849,Z 682.801,A -85,B 0,C 180,E1 -17281.414,E2 -17281.414} C_VEL
LIN {X 0,Y 284.689,Z 682.812,A -85,B 0,C 180,E1 -17287.091,E2 -17287.091} C_VEL
LIN {X 0,Y 284.56,Z 682.845,A -85,B 0,C 180,E1 -17289.956,E2 -17289.956} C_VEL
LIN {X 0,Y 284.472,Z 682.847,A -85,B 0,C 180,E1 -17294.304,E2 -17294.304} C_VEL
LIN {X 0,Y 284.419,Z 682.848,A -85,B 0,C 180,E1 -17297.249,E2 -17297.249} C_VEL
LIN {X 0,Y 284.378,Z 682.873,A -85,B 0,C 180,E1 -17300.009,E2 -17300.009} C_VEL
LIN {X 0,Y 283.739,Z 682.97,A -85,B 0,C 180,E1 -17301.191,E2 -17301.191} C_VEL
LIN {X 0,Y 280.861,Z 683.329,A -85,B 0,C 180,E1 -17303.117,E2 -17303.117} C_VEL
LIN {X 0,Y 278.409,Z 683.619,A -85,B 0,C 180,E1 -17304.681,E2 -17304.681} C_VEL
LIN {X 0,Y 277.375,Z 683.717,A -85,B 0,C 180,E1 -17305.895,E2 -17305.895} C_VEL
LIN {X 0,Y 277.302,Z 683.714,A -85,B 0,C 180,E1 -17306.306,E2 -17306.306} C_VEL
LIN {X 0,Y 277.267,Z 683.701,A -85,B 0,C 180,E1 -17310.482,E2 -17310.482} C_VEL
LIN {X 0,Y 277.31,Z 684.025,A -85,B 0,C 180,E1 -17313.247,E2 -17313.247} C_VEL
LIN {X 0,Y 277.709,Z 685.456,A -85,B 0,C 180,E1 -17313.832,E2 -17313.832} C_VEL
LIN {X 0,Y 280.781,Z 689.821,A -85,B 0,C 180,E1 -17314.984,E2 -17314.984} C_VEL
LIN {X 0,Y 282.638,Z 692.248,A -85,B 0,C 180,E1 -17315.618,E2 -17315.618} C_VEL
LIN {X 0,Y 287.075,Z 698.731,A -85,B 0,C 180,E1 -17317.09,E2 -17317.09} C_VEL
LIN {X 0,Y 290.925,Z 704.535,A -85,B 0,C 180,E1 -17318.301,E2 -17318.301} C_VEL
LIN {X 0,Y 296.99,Z 714.067,A -85,B 0,C 180,E1 -17320.099,E2 -17320.099} C_VEL
LIN {X 0,Y 304.839,Z 727.597,A -85,B 0,C 180,E1 -17322.273,E2 -17322.273} C_VEL
LIN {X 0,Y 312.499,Z 742.228,A -85,B 0,C 180,E1 -17324.258,E2 -17324.258} C_VEL
LIN {X 0,Y 320.634,Z 759.692,A -85,B 0,C 180,E1 -17326.251,E2 -17326.251} C_VEL
LIN {X 0,Y 321.662,Z 762.059,A -85,B 0,C 180,E1 -17326.496,E2 -17326.496} C_VEL
LIN {X 0,Y 315.465,Z 890.347,A -85,B 0,C 180,E1 -17329.346,E2 -17329.346} C_VEL
LIN {X 0,Y 314.381,Z 903.162,A -85,B 0,C 180,E1 -17329.746,E2 -17329.746} C_VEL
LIN {X 0,Y 312.852,Z 915.517,A -85,B 0,C 180,E1 -17330.245,E2 -17330.245} C_VEL
LIN {X 0,Y 310.989,Z 927.433,A -85,B 0,C 180,E1 -17330.851,E2 -17330.851} C_VEL
LIN {X 0,Y 308.806,Z 940.014,A -85,B 0,C 180,E1 -17331.673,E2 -17331.673} C_VEL
LIN {X 0,Y 306.073,Z 953.247,A -85,B 0,C 180,E1 -17332.728,E2 -17332.728} C_VEL
LIN {X 0,Y 303.119,Z 965.982,A -85,B 0,C 180,E1 -17333.962,E2 -17333.962} C_VEL
LIN {X 0,Y 300.225,Z 977.379,A -85,B 0,C 180,E1 -17335.275,E2 -17335.275} C_VEL
LIN {X 0,Y 297.283,Z 987.772,A -85,B 0,C 180,E1 -17336.658,E2 -17336.658} C_VEL
LIN {X 0,Y 294.218,Z 998.27,A -85,B 0,C 180,E1 -17338.298,E2 -17338.298} C_VEL
LIN {X 0,Y 291.33,Z 1007.65,A -85,B 0,C 180,E1 -17339.99,E2 -17339.99} C_VEL
LIN {X 0,Y 288.298,Z 1017.271,A -85,B 0,C 180,E1 -17342.014,E2 -17342.014} C_VEL
LIN {X 0,Y 285.544,Z 1025.795,A -85,B 0,C 180,E1 -17344.096,E2 -17344.096} C_VEL
LIN {X 0,Y 282.739,Z 1034.394,A -85,B 0,C 180,E1 -17346.566,E2 -17346.566} C_VEL
LIN {X 0,Y 280.837,Z 1040.829,A -85,B 0,C 180,E1 -17348.724,E2 -17348.724} C_VEL
LIN {X 0,Y 278.681,Z 1048.093,A -85,B 0,C 180,E1 -17351.626,E2 -17351.626} C_VEL
LIN {X 0,Y 277.467,Z 1052.748,A -85,B 0,C 180,E1 -17353.823,E2 -17353.823} C_VEL
LIN {X 0,Y 276.343,Z 1057.852,A -85,B 0,C 180,E1 -17356.769,E2 -17356.769} C_VEL
LIN {X 0,Y 275.609,Z 1061.855,A -85,B 0,C 180,E1 -17359.718,E2 -17359.718} C_VEL
LIN {X 0,Y 275.297,Z 1064.818,A -85,B 0,C 180,E1 -17362.667,E2 -17362.667} C_VEL
LIN {X 0,Y 275.228,Z 1066.379,A -85,B 0,C 180,E1 -17364.792,E2 -17364.792} C_VEL
LIN {X 0,Y 275.231,Z 1067.48,A -85,B 0,C 180,E1 -17367.073,E2 -17367.073} C_VEL
LIN {X 0,Y 275.275,Z 1067.97,A -85,B 0,C 180,E1 -17370,E2 -17370} C_VEL
LIN {X 0,Y 275.231,Z 1067.48,A -85,B 0,C 180,E1 -17372.927,E2 -17372.927} C_VEL
LIN {X 0,Y 275.235,Z 1066.007,A -85,B 0,C 180,E1 -17375.862,E2 -17375.862} C_VEL
LIN {X 0,Y 275.412,Z 1063.532,A -85,B 0,C 180,E1 -17378.807,E2 -17378.807} C_VEL
LIN {X 0,Y 276.15,Z 1058.942,A -85,B 0,C 180,E1 -17382.493,E2 -17382.493} C_VEL
LIN {X 0,Y 276.878,Z 1055.449,A -85,B 0,C 180,E1 -17384.704,E2 -17384.704} C_VEL
LIN {X 0,Y 278.222,Z 1049.715,A -85,B 0,C 180,E1 -17387.645,E2 -17387.645} C_VEL
LIN {X 0,Y 279.702,Z 1044.654,A -85,B 0,C 180,E1 -17389.828,E2 -17389.828} C_VEL
LIN {X 0,Y 282.031,Z 1036.886,A -85,B 0,C 180,E1 -17392.628,E2 -17392.628} C_VEL
LIN {X 0,Y 284.276,Z 1029.633,A -85,B 0,C 180,E1 -17394.852,E2 -17394.852} C_VEL
LIN {X 0,Y 286.851,Z 1021.666,A -85,B 0,C 180,E1 -17396.952,E2 -17396.952} C_VEL
LIN {X 0,Y 289.728,Z 1012.552,A -85,B 0,C 180,E1 -17399.021,E2 -17399.021} C_VEL
LIN {X 0,Y 292.454,Z 1003.987,A -85,B 0,C 180,E1 -17400.707,E2 -17400.707} C_VEL
LIN {X 0,Y 295.931,Z 992.121,A -85,B 0,C 180,E1 -17402.702,E2 -17402.702} C_VEL
LIN {X 0,Y 298.935,Z 981.961,A -85,B 0,C 180,E1 -17404.145,E2 -17404.145} C_VEL
LIN {X 0,Y 302.055,Z 970.296,A -85,B 0,C 180,E1 -17405.568,E2 -17405.568} C_VEL
LIN {X 0,Y 304.931,Z 958.272,A -85,B 0,C 180,E1 -17406.815,E2 -17406.815} C_VEL
LIN {X 0,Y 307.641,Z 945.957,A -85,B 0,C 180,E1 -17407.875,E2 -17407.875} C_VEL
LIN {X 0,Y 309.982,Z 933.414,A -85,B 0,C 180,E1 -17408.778,E2 -17408.778} C_VEL
LIN {X 0,Y 312.147,Z 919.99,A -85,B 0,C 180,E1 -17409.549,E2 -17409.549} C_VEL
LIN {X 0,Y 313.915,Z 907.077,A -85,B 0,C 180,E1 -17410.116,E2 -17410.116} C_VEL
LIN {X 0,Y 315.286,Z 893.794,A -85,B 0,C 180,E1 -17410.551,E2 -17410.551} C_VEL
LIN {X 0,Y 316.686,Z 865.473,A -85,B 0,C 180,E1 -17411.237,E2 -17411.237} C_VEL
LIN {X 0,Y 321.615,Z 763.08,A -85,B 0,C 180,E1 -17413.481,E2 -17413.481} C_VEL
LIN {X 0,Y 321.374,Z 761.351,A -85,B 0,C 180,E1 -17413.574,E2 -17413.574} C_VEL
LIN {X 0,Y 313.858,Z 745.015,A -85,B 0,C 180,E1 -17415.401,E2 -17415.401} C_VEL
LIN {X 0,Y 306.593,Z 730.837,A -85,B 0,C 180,E1 -17417.261,E2 -17417.261} C_VEL
LIN {X 0,Y 298.347,Z 716.327,A -85,B 0,C 180,E1 -17419.513,E2 -17419.513} C_VEL
LIN {X 0,Y 292.122,Z 706.37,A -85,B 0,C 180,E1 -17421.335,E2 -17421.335} C_VEL
LIN {X 0,Y 288.441,Z 700.793,A -85,B 0,C 180,E1 -17422.473,E2 -17422.473} C_VEL
LIN {X 0,Y 285.18,Z 695.928,A -85,B 0,C 180,E1 -17423.528,E2 -17423.528} C_VEL
LIN {X 0,Y 281.286,Z 690.383,A -85,B 0,C 180,E1 -17424.846,E2 -17424.846} C_VEL
LIN {X 0,Y 278.059,Z 686.225,A -85,B 0,C 180,E1 -17425.998,E2 -17425.998} C_VEL
LIN {X 0,Y 277.508,Z 684.903,A -85,B 0,C 180,E1 -17426.339,E2 -17426.339} C_VEL
LIN {X 0,Y 277.293,Z 683.855,A -85,B 0,C 180,E1 -17426.903,E2 -17426.903} C_VEL
LIN {X 0,Y 277.265,Z 683.686,A -85,B 0,C 180,E1 -17431.21,E2 -17431.21} C_VEL
LIN {X 0,Y 277.307,Z 683.736,A -85,B 0,C 180,E1 -17434.479,E2 -17434.479} C_VEL
LIN {X 0,Y 277.281,Z 683.738,A -85,B 0,C 180,E1 -17437.654,E2 -17437.654} C_VEL
LIN {X 0,Y 277.34,Z 683.739,A -85,B 0,C 180,E1 -17440.766,E2 -17440.766} C_VEL
LIN {X 0,Y 277.422,Z 683.733,A -85,B 0,C 180,E1 -17445.325,E2 -17445.325} C_VEL
LIN {X 0,Y 277.501,Z 683.729,A -85,B 0,C 180,E1 -17449.788,E2 -17449.788} C_VEL
LIN {X 0,Y 277.644,Z 683.688,A -85,B 0,C 180,E1 -17452.729,E2 -17452.729} C_VEL
LIN {X 0,Y 277.815,Z 683.675,A -85,B 0,C 180,E1 -17458.55,E2 -17458.55} C_VEL
LIN {X 0,Y 277.815,Z 683.671,A -85,B 0,C 180,E1 -17461.449,E2 -17461.449} C_VEL
LIN {X 0,Y 277.642,Z 683.69,A -85,B 0,C 180,E1 -17467.271,E2 -17467.271} C_VEL
LIN {X 0,Y 277.499,Z 683.731,A -85,B 0,C 180,E1 -17470.211,E2 -17470.211} C_VEL
LIN {X 0,Y 277.42,Z 683.733,A -85,B 0,C 180,E1 -17474.674,E2 -17474.674} C_VEL
LIN {X 0,Y 277.364,Z 683.738,A -85,B 0,C 180,E1 -17479.232,E2 -17479.232} C_VEL
LIN {X 0,Y 277.337,Z 683.745,A -85,B 0,C 180,E1 -17483.919,E2 -17483.919} C_VEL
LIN {X 0,Y 277.318,Z 683.687,A -85,B 0,C 180,E1 -17487.505,E2 -17487.505} C_VEL
LIN {X 0,Y 277.265,Z 683.702,A -85,B 0,C 180,E1 -17490.481,E2 -17490.481} C_VEL
LIN {X 0,Y 277.26,Z 683.855,A -85,B 0,C 180,E1 -17493.693,E2 -17493.693} C_VEL
LIN {X 0,Y 277.528,Z 685.054,A -85,B 0,C 180,E1 -17494.184,E2 -17494.184} C_VEL
LIN {X 0,Y 279.174,Z 687.745,A -85,B 0,C 180,E1 -17494.829,E2 -17494.829} C_VEL
LIN {X 0,Y 281.298,Z 689.53,A -85,B 0,C 180,E1 -17495.528,E2 -17495.528} C_VEL
LIN {X 0,Y 283.381,Z 692.768,A -85,B 0,C 180,E1 -17496.255,E2 -17496.255} C_VEL
LIN {X 0,Y 285.207,Z 694.646,A -85,B 0,C 180,E1 -17496.833,E2 -17496.833} C_VEL
LIN {X 0,Y 287.804,Z 698.321,A -85,B 0,C 180,E1 -17497.671,E2 -17497.671} C_VEL
LIN {X 0,Y 289.385,Z 700.227,A -85,B 0,C 180,E1 -17498.153,E2 -17498.153} C_VEL
LIN {X 0,Y 292.641,Z 704.135,A -85,B 0,C 180,E1 -17499.113,E2 -17499.113} C_VEL
LIN {X 0,Y 296.847,Z 709.123,A -85,B 0,C 180,E1 -17500.304,E2 -17500.304} C_VEL
LIN {X 0,Y 299.099,Z 711.565,A -85,B 0,C 180,E1 -17500.95,E2 -17500.95} C_VEL
LIN {X 0,Y 303.022,Z 715.627,A -85,B 0,C 180,E1 -17502.066,E2 -17502.066} C_VEL
LIN {X 0,Y 308.579,Z 721.364,A -85,B 0,C 180,E1 -17503.765,E2 -17503.765} C_VEL
LIN {X 0,Y 311.109,Z 723.777,A -85,B 0,C 180,E1 -17504.587,E2 -17504.587} C_VEL
LIN {X 0,Y 315.218,Z 727.936,A -85,B 0,C 180,E1 -17505.958,E2 -17505.958} C_VEL
LIN {X 0,Y 317.535,Z 730.198,A -85,B 0,C 180,E1 -17506.787,E2 -17506.787} C_VEL
LIN {X 0,Y 321.568,Z 734.275,A -85,B 0,C 180,E1 -17508.279,E2 -17508.279} C_VEL
LIN {X 0,Y 323.768,Z 736.497,A -85,B 0,C 180,E1 -17509.125,E2 -17509.125} C_VEL
LIN {X 0,Y 327.881,Z 740.598,A -85,B 0,C 180,E1 -17510.737,E2 -17510.737} C_VEL
LIN {X 0,Y 330.418,Z 743.225,A -85,B 0,C 180,E1 -17511.745,E2 -17511.745} C_VEL
LIN {X 0,Y 334.495,Z 747.033,A -85,B 0,C 180,E1 -17513.407,E2 -17513.407} C_VEL
LIN {X 0,Y 339.853,Z 752.438,A -85,B 0,C 180,E1 -17515.683,E2 -17515.683} C_VEL
LIN {X 0,Y 342.957,Z 755.077,A -85,B 0,C 180,E1 -17517.031,E2 -17517.031} C_VEL
LIN {X 0,Y 347.128,Z 759.214,A -85,B 0,C 180,E1 -17518.952,E2 -17518.952} C_VEL
LIN {X 0,Y 349.914,Z 761.542,A -85,B 0,C 180,E1 -17520.258,E2 -17520.258} C_VEL
LIN {X 0,Y 353.529,Z 765.244,A -85,B 0,C 180,E1 -17522.071,E2 -17522.071} C_VEL
LIN {X 0,Y 357.168,Z 768.123,A -85,B 0,C 180,E1 -17523.937,E2 -17523.937} C_VEL
LIN {X 0,Y 360.507,Z 771.647,A -85,B 0,C 180,E1 -17525.834,E2 -17525.834} C_VEL
LIN {X 0,Y 364.233,Z 774.269,A -85,B 0,C 180,E1 -17528.003,E2 -17528.003} C_VEL
LIN {X 0,Y 365.64,Z 775.678,A -85,B 0,C 180,E1 -17528.919,E2 -17528.919} C_VEL
LIN {X 0,Y 368.543,Z 778.638,A -85,B 0,C 180,E1 -17530.913,E2 -17530.913} C_VEL
LIN {X 0,Y 371.643,Z 780.812,A -85,B 0,C 180,E1 -17533.192,E2 -17533.192} C_VEL
LIN {X 0,Y 373.333,Z 781.859,A -85,B 0,C 180,E1 -17534.558,E2 -17534.558} C_VEL
LIN {X 0,Y 375.33,Z 784.344,A -85,B 0,C 180,E1 -17536.477,E2 -17536.477} C_VEL
LIN {X 0,Y 377.361,Z 786.218,A -85,B 0,C 180,E1 -17538.649,E2 -17538.649} C_VEL
LIN {X 0,Y 379.28,Z 787.37,A -85,B 0,C 180,E1 -17541.071,E2 -17541.071} C_VEL
LIN {X 0,Y 380.852,Z 788.091,A -85,B 0,C 180,E1 -17543.643,E2 -17543.643} C_VEL
LIN {X 0,Y 381.72,Z 788.692,A -85,B 0,C 180,E1 -17545.777,E2 -17545.777} C_VEL
LIN {X 0,Y 382.275,Z 788.889,A -85,B 0,C 180,E1 -17547.893,E2 -17547.893} C_VEL
LIN {X 0,Y 382.474,Z 788.96,A -85,B 0,C 180,E1 -17550,E2 -17550} C_VEL
LIN {X 0,Y 382.275,Z 788.89,A -85,B 0,C 180,E1 -17552.107,E2 -17552.107} C_VEL
LIN {X 0,Y 381.573,Z 788.548,A -85,B 0,C 180,E1 -17554.668,E2 -17554.668} C_VEL
LIN {X 0,Y 380.355,Z 787.915,A -85,B 0,C 180,E1 -17557.251,E2 -17557.251} C_VEL
LIN {X 0,Y 378.388,Z 786.897,A -85,B 0,C 180,E1 -17560.139,E2 -17560.139} C_VEL
LIN {X 0,Y 376.234,Z 785.268,A -85,B 0,C 180,E1 -17562.581,E2 -17562.581} C_VEL
LIN {X 0,Y 374.021,Z 782.825,A -85,B 0,C 180,E1 -17564.797,E2 -17564.797} C_VEL
LIN {X 0,Y 372.753,Z 781.35,A -85,B 0,C 180,E1 -17565.938,E2 -17565.938} C_VEL
LIN {X 0,Y 369.831,Z 779.648,A -85,B 0,C 180,E1 -17568.167,E2 -17568.167} C_VEL
LIN {X 0,Y 366.608,Z 776.783,A -85,B 0,C 180,E1 -17570.427,E2 -17570.427} C_VEL
LIN {X 0,Y 364.46,Z 774.388,A -85,B 0,C 180,E1 -17571.854,E2 -17571.854} C_VEL
LIN {X 0,Y 360.507,Z 771.649,A -85,B 0,C 180,E1 -17574.166,E2 -17574.166} C_VEL
LIN {X 0,Y 356.126,Z 767.156,A -85,B 0,C 180,E1 -17576.612,E2 -17576.612} C_VEL
LIN {X 0,Y 352.465,Z 764.267,A -85,B 0,C 180,E1 -17578.469,E2 -17578.469} C_VEL
LIN {X 0,Y 348.724,Z 760.418,A -85,B 0,C 180,E1 -17580.318,E2 -17580.318} C_VEL
LIN {X 0,Y 344.582,Z 756.866,A -85,B 0,C 180,E1 -17582.214,E2 -17582.214} C_VEL
LIN {X 0,Y 341.721,Z 753.9,A -85,B 0,C 180,E1 -17583.509,E2 -17583.509} C_VEL
LIN {X 0,Y 337.466,Z 750.161,A -85,B 0,C 180,E1 -17585.34,E2 -17585.34} C_VEL
LIN {X 0,Y 334.497,Z 747.035,A -85,B 0,C 180,E1 -17586.593,E2 -17586.593} C_VEL
LIN {X 0,Y 330.419,Z 743.228,A -85,B 0,C 180,E1 -17588.255,E2 -17588.255} C_VEL
LIN {X 0,Y 327.883,Z 740.584,A -85,B 0,C 180,E1 -17589.264,E2 -17589.264} C_VEL
LIN {X 0,Y 323.898,Z 736.647,A -85,B 0,C 180,E1 -17590.823,E2 -17590.823} C_VEL
LIN {X 0,Y 321.628,Z 734.34,A -85,B 0,C 180,E1 -17591.699,E2 -17591.699} C_VEL
LIN {X 0,Y 317.641,Z 730.323,A -85,B 0,C 180,E1 -17593.169,E2 -17593.169} C_VEL
LIN {X 0,Y 315.082,Z 727.786,A -85,B 0,C 180,E1 -17594.09,E2 -17594.09} C_VEL
LIN {X 0,Y 311.104,Z 723.79,A -85,B 0,C 180,E1 -17595.414,E2 -17595.414} C_VEL
LIN {X 0,Y 305.671,Z 718.56,A -85,B 0,C 180,E1 -17597.108,E2 -17597.108} C_VEL
LIN {X 0,Y 303.023,Z 715.617,A -85,B 0,C 180,E1 -17597.934,E2 -17597.934} C_VEL
LIN {X 0,Y 299.102,Z 711.535,A -85,B 0,C 180,E1 -17599.051,E2 -17599.051} C_VEL
LIN {X 0,Y 296.309,Z 708.575,A -85,B 0,C 180,E1 -17599.846,E2 -17599.846} C_VEL
LIN {X 0,Y 291.716,Z 703.211,A -85,B 0,C 180,E1 -17601.148,E2 -17601.148} C_VEL
LIN {X 0,Y 288.094,Z 698.603,A -85,B 0,C 180,E1 -17602.242,E2 -17602.242} C_VEL
LIN {X 0,Y 285.441,Z 695.073,A -85,B 0,C 180,E1 -17603.086,E2 -17603.086} C_VEL
LIN {X 0,Y 284.467,Z 693.786,A -85,B 0,C 180,E1 -17603.403,E2 -17603.403} C_VEL
LIN {X 0,Y 282.055,Z 690.974,A -85,B 0,C 180,E1 -17604.194,E2 -17604.194} C_VEL
LIN {X 0,Y 281.065,Z 689.16,A -85,B 0,C 180,E1 -17604.555,E2 -17604.555} C_VEL
LIN {X 0,Y 278.62,Z 687.072,A -85,B 0,C 180,E1 -17605.367,E2 -17605.367} C_VEL
LIN {X 0,Y 277.417,Z 684.683,A -85,B 0,C 180,E1 -17605.91,E2 -17605.91} C_VEL
LIN {X 0,Y 277.256,Z 683.797,A -85,B 0,C 180,E1 -17606.406,E2 -17606.406} C_VEL
LIN {X 0,Y 277.255,Z 683.703,A -85,B 0,C 180,E1 -17609.538,E2 -17609.538} C_VEL
LIN {X 0,Y 277.351,Z 683.688,A -85,B 0,C 180,E1 -17612.864,E2 -17612.864} C_VEL
LIN {X 0,Y 277.337,Z 683.745,A -85,B 0,C 180,E1 -17616.081,E2 -17616.081} C_VEL
LIN {X 0,Y 277.364,Z 683.738,A -85,B 0,C 180,E1 -17620.768,E2 -17620.768} C_VEL
LIN {X 0,Y 277.42,Z 683.732,A -85,B 0,C 180,E1 -17625.326,E2 -17625.326} C_VEL
LIN {X 0,Y 277.499,Z 683.729,A -85,B 0,C 180,E1 -17629.789,E2 -17629.789} C_VEL
LIN {X 0,Y 277.64,Z 683.689,A -85,B 0,C 180,E1 -17632.729,E2 -17632.729} C_VEL
LIN {X 0,Y 277.815,Z 683.672,A -85,B 0,C 180,E1 -17638.551,E2 -17638.551} C_VEL
LIN {X 0,Y 277.815,Z 683.676,A -85,B 0,C 180,E1 -17641.45,E2 -17641.45} C_VEL
LIN {X 0,Y 277.644,Z 683.688,A -85,B 0,C 180,E1 -17647.271,E2 -17647.271} C_VEL
LIN {X 0,Y 277.501,Z 683.727,A -85,B 0,C 180,E1 -17650.212,E2 -17650.212} C_VEL
LIN {X 0,Y 277.422,Z 683.73,A -85,B 0,C 180,E1 -17654.675,E2 -17654.675} C_VEL
LIN {X 0,Y 277.34,Z 683.739,A -85,B 0,C 180,E1 -17659.234,E2 -17659.234} C_VEL
LIN {X 0,Y 277.313,Z 683.75,A -85,B 0,C 180,E1 -17664.171,E2 -17664.171} C_VEL
LIN {X 0,Y 277.302,Z 683.714,A -85,B 0,C 180,E1 -17666.306,E2 -17666.306} C_VEL
LIN {X 0,Y 276.629,Z 683.78,A -85,B 0,C 180,E1 -17667.113,E2 -17667.113} C_VEL
LIN {X 0,Y 273.751,Z 684.124,A -85,B 0,C 180,E1 -17668.376,E2 -17668.376} C_VEL
LIN {X 0,Y 270.858,Z 684.507,A -85,B 0,C 180,E1 -17669.665,E2 -17669.665} C_VEL
LIN {X 0,Y 270.197,Z 684.645,A -85,B 0,C 180,E1 -17670.501,E2 -17670.501} C_VEL
LIN {X 0,Y 270.263,Z 684.959,A -85,B 0,C 180,E1 -17671.185,E2 -17671.185} C_VEL
LIN {X 0,Y 270.631,Z 686.353,A -85,B 0,C 180,E1 -17671.618,E2 -17671.618} C_VEL
LIN {X 0,Y 272.419,Z 688.964,A -85,B 0,C 180,E1 -17672.366,E2 -17672.366} C_VEL
LIN {X 0,Y 274.529,Z 690.85,A -85,B 0,C 180,E1 -17673.137,E2 -17673.137} C_VEL
LIN {X 0,Y 278.151,Z 695.937,A -85,B 0,C 180,E1 -17674.481,E2 -17674.481} C_VEL
LIN {X 0,Y 279.806,Z 698.254,A -85,B 0,C 180,E1 -17675.069,E2 -17675.069} C_VEL
LIN {X 0,Y 283.746,Z 704.014,A -85,B 0,C 180,E1 -17676.419,E2 -17676.419} C_VEL
LIN {X 0,Y 290.397,Z 714.302,A -85,B 0,C 180,E1 -17678.549,E2 -17678.549} C_VEL
LIN {X 0,Y 297.177,Z 725.794,A -85,B 0,C 180,E1 -17680.568,E2 -17680.568} C_VEL
LIN {X 0,Y 303.816,Z 737.907,A -85,B 0,C 180,E1 -17682.416,E2 -17682.416} C_VEL
LIN {X 0,Y 310.935,Z 752.269,A -85,B 0,C 180,E1 -17684.288,E2 -17684.288} C_VEL
LIN {X 0,Y 316.375,Z 764.38,A -85,B 0,C 180,E1 -17685.659,E2 -17685.659} C_VEL
LIN {X 0,Y 310.136,Z 889.931,A -85,B 0,C 180,E1 -17688.486,E2 -17688.486} C_VEL
LIN {X 0,Y 308.995,Z 902.957,A -85,B 0,C 180,E1 -17688.895,E2 -17688.895} C_VEL
LIN {X 0,Y 307.299,Z 916.057,A -85,B 0,C 180,E1 -17689.432,E2 -17689.432} C_VEL
LIN {X 0,Y 305.302,Z 928.424,A -85,B 0,C 180,E1 -17690.084,E2 -17690.084} C_VEL
LIN {X 0,Y 303.245,Z 939.808,A -85,B 0,C 180,E1 -17690.837,E2 -17690.837} C_VEL
LIN {X 0,Y 300.425,Z 953.04,A -85,B 0,C 180,E1 -17691.904,E2 -17691.904} C_VEL
LIN {X 0,Y 297.377,Z 965.775,A -85,B 0,C 180,E1 -17693.153,E2 -17693.153} C_VEL
LIN {X 0,Y 294.513,Z 976.577,A -85,B 0,C 180,E1 -17694.401,E2 -17694.401} C_VEL
LIN {X 0,Y 291.348,Z 987.566,A -85,B 0,C 180,E1 -17695.887,E2 -17695.887} C_VEL
LIN {X 0,Y 288.113,Z 998.061,A -85,B 0,C 180,E1 -17697.545,E2 -17697.545} C_VEL
LIN {X 0,Y 285.17,Z 1007.332,A -85,B 0,C 180,E1 -17699.245,E2 -17699.245} C_VEL
LIN {X 0,Y 281.943,Z 1017.062,A -85,B 0,C 180,E1 -17701.326,E2 -17701.326} C_VEL
LIN {X 0,Y 279.054,Z 1025.585,A -85,B 0,C 180,E1 -17703.447,E2 -17703.447} C_VEL
LIN {X 0,Y 276.133,Z 1034.186,A -85,B 0,C 180,E1 -17705.97,E2 -17705.97} C_VEL
LIN {X 0,Y 274.131,Z 1040.621,A -85,B 0,C 180,E1 -17708.178,E2 -17708.178} C_VEL
LIN {X 0,Y 271.851,Z 1047.885,A -85,B 0,C 180,E1 -17711.147,E2 -17711.147} C_VEL
LIN {X 0,Y 270.552,Z 1052.539,A -85,B 0,C 180,E1 -17713.397,E2 -17713.397} C_VEL
LIN {X 0,Y 269.341,Z 1057.643,A -85,B 0,C 180,E1 -17716.418,E2 -17716.418} C_VEL
LIN {X 0,Y 268.563,Z 1061.648,A -85,B 0,C 180,E1 -17719.445,E2 -17719.445} C_VEL
LIN {X 0,Y 268.228,Z 1064.611,A -85,B 0,C 180,E1 -17722.472,E2 -17722.472} C_VEL
LIN {X 0,Y 268.13,Z 1066.284,A -85,B 0,C 180,E1 -17724.888,E2 -17724.888} C_VEL
LIN {X 0,Y 268.142,Z 1067.275,A -85,B 0,C 180,E1 -17726.995,E2 -17726.995} C_VEL
LIN {X 0,Y 268.199,Z 1067.765,A -85,B 0,C 180,E1 -17730,E2 -17730} C_VEL
LIN {X 0,Y 268.142,Z 1067.275,A -85,B 0,C 180,E1 -17733.005,E2 -17733.005} C_VEL
LIN {X 0,Y 268.145,Z 1065.8,A -85,B 0,C 180,E1 -17736.018,E2 -17736.018} C_VEL
LIN {X 0,Y 268.353,Z 1063.326,A -85,B 0,C 180,E1 -17739.04,E2 -17739.04} C_VEL
LIN {X 0,Y 269.127,Z 1058.734,A -85,B 0,C 180,E1 -17742.824,E2 -17742.824} C_VEL
LIN {X 0,Y 269.918,Z 1055.24,A -85,B 0,C 180,E1 -17745.092,E2 -17745.092} C_VEL
LIN {X 0,Y 271.375,Z 1049.507,A -85,B 0,C 180,E1 -17748.105,E2 -17748.105} C_VEL
LIN {X 0,Y 272.952,Z 1044.446,A -85,B 0,C 180,E1 -17750.34,E2 -17750.34} C_VEL
LIN {X 0,Y 275.415,Z 1036.484,A -85,B 0,C 180,E1 -17753.272,E2 -17753.272} C_VEL
LIN {X 0,Y 277.757,Z 1029.425,A -85,B 0,C 180,E1 -17755.476,E2 -17755.476} C_VEL
LIN {X 0,Y 280.454,Z 1021.457,A -85,B 0,C 180,E1 -17757.619,E2 -17757.619} C_VEL
LIN {X 0,Y 283.469,Z 1012.345,A -85,B 0,C 180,E1 -17759.725,E2 -17759.725} C_VEL
LIN {X 0,Y 286.303,Z 1003.779,A -85,B 0,C 180,E1 -17761.441,E2 -17761.441} C_VEL
LIN {X 0,Y 289.907,Z 991.913,A -85,B 0,C 180,E1 -17763.47,E2 -17763.47} C_VEL
LIN {X 0,Y 293.052,Z 981.755,A -85,B 0,C 180,E1 -17764.929,E2 -17764.929} C_VEL
LIN {X 0,Y 296.249,Z 970.088,A -85,B 0,C 180,E1 -17766.375,E2 -17766.375} C_VEL
LIN {X 0,Y 299.246,Z 958.065,A -85,B 0,C 180,E1 -17767.634,E2 -17767.634} C_VEL
LIN {X 0,Y 302.034,Z 945.75,A -85,B 0,C 180,E1 -17768.707,E2 -17768.707} C_VEL
LIN {X 0,Y 304.468,Z 933.209,A -85,B 0,C 180,E1 -17769.617,E2 -17769.617} C_VEL
LIN {X 0,Y 306.703,Z 919.785,A -85,B 0,C 180,E1 -17770.394,E2 -17770.394} C_VEL
LIN {X 0,Y 308.515,Z 906.872,A -85,B 0,C 180,E1 -17770.967,E2 -17770.967} C_VEL
LIN {X 0,Y 309.942,Z 893.495,A -85,B 0,C 180,E1 -17771.405,E2 -17771.405} C_VEL
LIN {X 0,Y 311.36,Z 865.718,A -85,B 0,C 180,E1 -17772.089,E2 -17772.089} C_VEL
LIN {X 0,Y 316.399,Z 764.328,A -85,B 0,C 180,E1 -17774.339,E2 -17774.339} C_VEL
LIN {X 0,Y 307.492,Z 745.064,A -85,B 0,C 180,E1 -17776.607,E2 -17776.607} C_VEL
LIN {X 0,Y 299.912,Z 730.648,A -85,B 0,C 180,E1 -17778.657,E2 -17778.657} C_VEL
LIN {X 0,Y 292.776,Z 718.106,A -85,B 0,C 180,E1 -17780.73,E2 -17780.73} C_VEL
LIN {X 0,Y 285.963,Z 707.386,A -85,B 0,C 180,E1 -17782.851,E2 -17782.851} C_VEL
LIN {X 0,Y 282.051,Z 701.527,A -85,B 0,C 180,E1 -17784.152,E2 -17784.152} C_VEL
LIN {X 0,Y 278.374,Z 696.213,A -85,B 0,C 180,E1 -17785.44,E2 -17785.44} C_VEL
LIN {X 0,Y 274.667,Z 691.12,A -85,B 0,C 180,E1 -17786.807,E2 -17786.807} C_VEL
LIN {X 0,Y 273.554,Z 689.833,A -85,B 0,C 180,E1 -17787.223,E2 -17787.223} C_VEL
LIN {X 0,Y 271.37,Z 687.739,A -85,B 0,C 180,E1 -17788.042,E2 -17788.042} C_VEL
LIN {X 0,Y 270.297,Z 685.268,A -85,B 0,C 180,E1 -17788.666,E2 -17788.666} C_VEL
LIN {X 0,Y 270.219,Z 684.682,A -85,B 0,C 180,E1 -17789.122,E2 -17789.122} C_VEL
LIN {X 0,Y 270.259,Z 684.562,A -85,B 0,C 180,E1 -17792.145,E2 -17792.145} C_VEL
LIN {X 0,Y 270.272,Z 684.632,A -85,B 0,C 180,E1 -17795.519,E2 -17795.519} C_VEL
LIN {X 0,Y 270.296,Z 684.625,A -85,B 0,C 180,E1 -17800.244,E2 -17800.244} C_VEL
LIN {X 0,Y 270.39,Z 684.615,A -85,B 0,C 180,E1 -17804.934,E2 -17804.934} C_VEL
LIN {X 0,Y 270.436,Z 684.61,A -85,B 0,C 180,E1 -17809.518,E2 -17809.518} C_VEL
LIN {X 0,Y 270.602,Z 684.563,A -85,B 0,C 180,E1 -17812.538,E2 -17812.538} C_VEL
LIN {X 0,Y 270.781,Z 684.549,A -85,B 0,C 180,E1 -17818.512,E2 -17818.512} C_VEL
LIN {X 0,Y 270.781,Z 684.546,A -85,B 0,C 180,E1 -17821.487,E2 -17821.487} C_VEL
LIN {X 0,Y 270.601,Z 684.566,A -85,B 0,C 180,E1 -17827.461,E2 -17827.461} C_VEL
LIN {X 0,Y 270.434,Z 684.61,A -85,B 0,C 180,E1 -17830.481,E2 -17830.481} C_VEL
LIN {X 0,Y 270.389,Z 684.615,A -85,B 0,C 180,E1 -17835.065,E2 -17835.065} C_VEL
LIN {X 0,Y 270.319,Z 684.624,A -85,B 0,C 180,E1 -17839.754,E2 -17839.754} C_VEL
LIN {X 0,Y 270.272,Z 684.633,A -85,B 0,C 180,E1 -17844.585,E2 -17844.585} C_VEL
LIN {X 0,Y 270.263,Z 684.56,A -85,B 0,C 180,E1 -17847.909,E2 -17847.909} C_VEL
LIN {X 0,Y 270.222,Z 684.77,A -85,B 0,C 180,E1 -17851.452,E2 -17851.452} C_VEL
LIN {X 0,Y 270.496,Z 685.982,A -85,B 0,C 180,E1 -17851.963,E2 -17851.963} C_VEL
LIN {X 0,Y 272.053,Z 688.573,A -85,B 0,C 180,E1 -17852.633,E2 -17852.633} C_VEL
LIN {X 0,Y 274.49,Z 690.659,A -85,B 0,C 180,E1 -17853.523,E2 -17853.523} C_VEL
LIN {X 0,Y 276.461,Z 693.743,A -85,B 0,C 180,E1 -17854.279,E2 -17854.279} C_VEL
LIN {X 0,Y 278.604,Z 695.897,A -85,B 0,C 180,E1 -17855.021,E2 -17855.021} C_VEL
LIN {X 0,Y 281.311,Z 699.519,A -85,B 0,C 180,E1 -17855.961,E2 -17855.961} C_VEL
LIN {X 0,Y 282.556,Z 701.102,A -85,B 0,C 180,E1 -17856.377,E2 -17856.377} C_VEL
LIN {X 0,Y 286.965,Z 706.957,A -85,B 0,C 180,E1 -17857.8,E2 -17857.8} C_VEL
LIN {X 0,Y 294.272,Z 715.448,A -85,B 0,C 180,E1 -17859.93,E2 -17859.93} C_VEL
LIN {X 0,Y 300.119,Z 721.626,A -85,B 0,C 180,E1 -17861.575,E2 -17861.575} C_VEL
LIN {X 0,Y 306.205,Z 727.729,A -85,B 0,C 180,E1 -17863.39,E2 -17863.39} C_VEL
LIN {X 0,Y 308.866,Z 730.27,A -85,B 0,C 180,E1 -17864.222,E2 -17864.222} C_VEL
LIN {X 0,Y 313.296,Z 734.592,A -85,B 0,C 180,E1 -17865.677,E2 -17865.677} C_VEL
LIN {X 0,Y 315.918,Z 737.235,A -85,B 0,C 180,E1 -17866.596,E2 -17866.596} C_VEL
LIN {X 0,Y 320.229,Z 741.321,A -85,B 0,C 180,E1 -17868.159,E2 -17868.159} C_VEL
LIN {X 0,Y 325.239,Z 746.52,A -85,B 0,C 180,E1 -17870.096,E2 -17870.096} C_VEL
LIN {X 0,Y 327.845,Z 749.002,A -85,B 0,C 180,E1 -17871.127,E2 -17871.127} C_VEL
LIN {X 0,Y 332.088,Z 753.205,A -85,B 0,C 180,E1 -17872.835,E2 -17872.835} C_VEL
LIN {X 0,Y 334.19,Z 755.15,A -85,B 0,C 180,E1 -17873.701,E2 -17873.701} C_VEL
LIN {X 0,Y 338.69,Z 759.496,A -85,B 0,C 180,E1 -17875.601,E2 -17875.601} C_VEL
LIN {X 0,Y 341.447,Z 761.923,A -85,B 0,C 180,E1 -17876.801,E2 -17876.801} C_VEL
LIN {X 0,Y 345.766,Z 766.052,A -85,B 0,C 180,E1 -17878.756,E2 -17878.756} C_VEL
LIN {X 0,Y 348.621,Z 768.535,A -85,B 0,C 180,E1 -17880.094,E2 -17880.094} C_VEL
LIN {X 0,Y 352.388,Z 772.293,A -85,B 0,C 180,E1 -17881.972,E2 -17881.972} C_VEL
LIN {X 0,Y 355.821,Z 774.954,A -85,B 0,C 180,E1 -17883.717,E2 -17883.717} C_VEL
LIN {X 0,Y 359.287,Z 778.557,A -85,B 0,C 180,E1 -17885.662,E2 -17885.662} C_VEL
LIN {X 0,Y 363.062,Z 781.2,A -85,B 0,C 180,E1 -17887.839,E2 -17887.839} C_VEL
LIN {X 0,Y 364.413,Z 782.53,A -85,B 0,C 180,E1 -17888.718,E2 -17888.718} C_VEL
LIN {X 0,Y 367.267,Z 785.423,A -85,B 0,C 180,E1 -17890.634,E2 -17890.634} C_VEL
LIN {X 0,Y 370.28,Z 787.638,A -85,B 0,C 180,E1 -17892.835,E2 -17892.835} C_VEL
LIN {X 0,Y 372.28,Z 788.877,A -85,B 0,C 180,E1 -17894.423,E2 -17894.423} C_VEL
LIN {X 0,Y 374.599,Z 791.626,A -85,B 0,C 180,E1 -17896.631,E2 -17896.631} C_VEL
LIN {X 0,Y 376.81,Z 793.52,A -85,B 0,C 180,E1 -17899.045,E2 -17899.045} C_VEL
LIN {X 0,Y 378.687,Z 794.537,A -85,B 0,C 180,E1 -17901.462,E2 -17901.462} C_VEL
LIN {X 0,Y 380.176,Z 795.261,A -85,B 0,C 180,E1 -17904.09,E2 -17904.09} C_VEL
LIN {X 0,Y 380.849,Z 795.737,A -85,B 0,C 180,E1 -17905.767,E2 -17905.767} C_VEL
LIN {X 0,Y 381.41,Z 795.935,A -85,B 0,C 180,E1 -17907.888,E2 -17907.888} C_VEL
LIN {X 0,Y 381.609,Z 796.007,A -85,B 0,C 180,E1 -17910,E2 -17910} C_VEL
LIN {X 0,Y 381.41,Z 795.937,A -85,B 0,C 180,E1 -17912.112,E2 -17912.112} C_VEL
LIN {X 0,Y 380.62,Z 795.518,A -85,B 0,C 180,E1 -17914.946,E2 -17914.946} C_VEL
LIN {X 0,Y 379.368,Z 794.872,A -85,B 0,C 180,E1 -17917.451,E2 -17917.451} C_VEL
LIN {X 0,Y 377.496,Z 793.942,A -85,B 0,C 180,E1 -17920.163,E2 -17920.163} C_VEL
LIN {X 0,Y 375.328,Z 792.313,A -85,B 0,C 180,E1 -17922.612,E2 -17922.612} C_VEL
LIN {X 0,Y 373.089,Z 789.911,A -85,B 0,C 180,E1 -17924.834,E2 -17924.834} C_VEL
LIN {X 0,Y 371.709,Z 788.328,A -85,B 0,C 180,E1 -17926.063,E2 -17926.063} C_VEL
LIN {X 0,Y 368.634,Z 786.532,A -85,B 0,C 180,E1 -17928.377,E2 -17928.377} C_VEL
LIN {X 0,Y 365.377,Z 783.617,A -85,B 0,C 180,E1 -17930.659,E2 -17930.659} C_VEL
LIN {X 0,Y 363.234,Z 781.281,A -85,B 0,C 180,E1 -17932.061,E2 -17932.061} C_VEL
LIN {X 0,Y 359.292,Z 778.531,A -85,B 0,C 180,E1 -17934.337,E2 -17934.337} C_VEL
LIN {X 0,Y 355.557,Z 774.68,A -85,B 0,C 180,E1 -17936.422,E2 -17936.422} C_VEL
LIN {X 0,Y 351.138,Z 771.154,A -85,B 0,C 180,E1 -17938.663,E2 -17938.663} C_VEL
LIN {X 0,Y 347.158,Z 767.136,A -85,B 0,C 180,E1 -17940.596,E2 -17940.596} C_VEL
LIN {X 0,Y 343.012,Z 763.585,A -85,B 0,C 180,E1 -17942.492,E2 -17942.492} C_VEL
LIN {X 0,Y 339.901,Z 760.444,A -85,B 0,C 180,E1 -17943.884,E2 -17943.884} C_VEL
LIN {X 0,Y 335.533,Z 756.566,A -85,B 0,C 180,E1 -17945.74,E2 -17945.74} C_VEL
LIN {X 0,Y 332.63,Z 753.602,A -85,B 0,C 180,E1 -17946.956,E2 -17946.956} C_VEL
LIN {X 0,Y 328.251,Z 749.49,A -85,B 0,C 180,E1 -17948.71,E2 -17948.71} C_VEL
LIN {X 0,Y 325.789,Z 746.924,A -85,B 0,C 180,E1 -17949.697,E2 -17949.697} C_VEL
LIN {X 0,Y 321.518,Z 742.715,A -85,B 0,C 180,E1 -17951.346,E2 -17951.346} C_VEL
LIN {X 0,Y 318.728,Z 740.023,A -85,B 0,C 180,E1 -17952.396,E2 -17952.396} C_VEL
LIN {X 0,Y 313.297,Z 734.575,A -85,B 0,C 180,E1 -17954.324,E2 -17954.324} C_VEL
LIN {X 0,Y 308.943,Z 730.368,A -85,B 0,C 180,E1 -17955.752,E2 -17955.752} C_VEL
LIN {X 0,Y 306.196,Z 727.748,A -85,B 0,C 180,E1 -17956.609,E2 -17956.609} C_VEL
LIN {X 0,Y 301.848,Z 723.294,A -85,B 0,C 180,E1 -17957.934,E2 -17957.934} C_VEL
LIN {X 0,Y 296.283,Z 717.643,A -85,B 0,C 180,E1 -17959.507,E2 -17959.507} C_VEL
LIN {X 0,Y 290.508,Z 711.209,A -85,B 0,C 180,E1 -17961.136,E2 -17961.136} C_VEL
LIN {X 0,Y 286.021,Z 705.532,A -85,B 0,C 180,E1 -17962.504,E2 -17962.504} C_VEL
LIN {X 0,Y 282.335,Z 700.724,A -85,B 0,C 180,E1 -17963.7,E2 -17963.7} C_VEL
LIN {X 0,Y 278.818,Z 696.263,A -85,B 0,C 180,E1 -17964.9,E2 -17964.9} C_VEL
LIN {X 0,Y 277.936,Z 695.083,A -85,B 0,C 180,E1 -17965.214,E2 -17965.214} C_VEL
LIN {X 0,Y 275.342,Z 692.278,A -85,B 0,C 180,E1 -17966.134,E2 -17966.134} C_VEL
LIN {X 0,Y 274.009,Z 690.065,A -85,B 0,C 180,E1 -17966.658,E2 -17966.658} C_VEL
LIN {X 0,Y 271.633,Z 688.085,A -85,B 0,C 180,E1 -17967.53,E2 -17967.53} C_VEL
LIN {X 0,Y 270.322,Z 685.365,A -85,B 0,C 180,E1 -17968.233,E2 -17968.233} C_VEL
LIN {X 0,Y 270.201,Z 684.688,A -85,B 0,C 180,E1 -17968.655,E2 -17968.655} C_VEL
LIN {X 0,Y 270.257,Z 684.561,A -85,B 0,C 180,E1 -17972.146,E2 -17972.146} C_VEL
LIN {X 0,Y 270.275,Z 684.633,A -85,B 0,C 180,E1 -17975.517,E2 -17975.517} C_VEL
LIN {X 0,Y 270.319,Z 684.624,A -85,B 0,C 180,E1 -17980.246,E2 -17980.246} C_VEL
LIN {X 0,Y 270.389,Z 684.614,A -85,B 0,C 180,E1 -17984.935,E2 -17984.935} C_VEL
LIN {X 0,Y 270.434,Z 684.608,A -85,B 0,C 180,E1 -17989.519,E2 -17989.519} C_VEL
LIN {X 0,Y 270.599,Z 684.564,A -85,B 0,C 180,E1 -17992.539,E2 -17992.539} C_VEL
LIN {X 0,Y 270.781,Z 684.547,A -85,B 0,C 180,E1 -17998.513,E2 -17998.513} C_VEL
LIN {X 0,Y 270.781,Z 684.551,A -85,B 0,C 180,E1 -18001.488,E2 -18001.488} C_VEL
LIN {X 0,Y 270.602,Z 684.563,A -85,B 0,C 180,E1 -18007.462,E2 -18007.462} C_VEL
LIN {X 0,Y 270.436,Z 684.608,A -85,B 0,C 180,E1 -18010.482,E2 -18010.482} C_VEL
LIN {X 0,Y 270.39,Z 684.612,A -85,B 0,C 180,E1 -18015.066,E2 -18015.066} C_VEL
LIN {X 0,Y 270.296,Z 684.624,A -85,B 0,C 180,E1 -18019.756,E2 -18019.756} C_VEL
LIN {X 0,Y 270.269,Z 684.633,A -85,B 0,C 180,E1 -18024.586,E2 -18024.586} C_VEL
LIN {X 0,Y 270.265,Z 684.56,A -85,B 0,C 180,E1 -18027.91,E2 -18027.91} C_VEL
LIN {X 0,Y 270.197,Z 684.645,A -85,B 0,C 180,E1 -18030.501,E2 -18030.501} C_VEL
LIN {X 0,Y 270.503,Z 685.342,A -85,B 0,C 180,E1 -18031.17,E2 -18031.17} C_VEL
LIN {X 0,Y 271.425,Z 687.534,A -85,B 0,C 180,E1 -18031.912,E2 -18031.912} C_VEL
LIN {X 0,Y 273.075,Z 691.779,A -85,B 0,C 180,E1 -18032.715,E2 -18032.715} C_VEL
LIN {X 0,Y 276.201,Z 702.04,A -85,B 0,C 180,E1 -18034.158,E2 -18034.158} C_VEL
LIN {X 0,Y 277.963,Z 705.743,A -85,B 0,C 180,E1 -18034.859,E2 -18034.859} C_VEL
LIN {X 0,Y 278.394,Z 706.366,A -85,B 0,C 180,E1 -18035.013,E2 -18035.013} C_VEL
LIN {X 0,Y 280.866,Z 710.024,A -85,B 0,C 180,E1 -18035.877,E2 -18035.877} C_VEL
LIN {X 0,Y 287.244,Z 720.075,A -85,B 0,C 180,E1 -18037.988,E2 -18037.988} C_VEL
LIN {X 0,Y 293.455,Z 730.746,A -85,B 0,C 180,E1 -18039.903,E2 -18039.903} C_VEL
LIN {X 0,Y 300.08,Z 743.092,A -85,B 0,C 180,E1 -18041.817,E2 -18041.817} C_VEL
LIN {X 0,Y 306.789,Z 756.884,A -85,B 0,C 180,E1 -18043.647,E2 -18043.647} C_VEL
LIN {X 0,Y 311.171,Z 766.83,A -85,B 0,C 180,E1 -18044.8,E2 -18044.8} C_VEL
LIN {X 0,Y 307.023,Z 848.092,A -85,B 0,C 180,E1 -18046.63,E2 -18046.63} C_VEL
LIN {X 0,Y 304.734,Z 891.076,A -85,B 0,C 180,E1 -18047.637,E2 -18047.637} C_VEL
LIN {X 0,Y 303.566,Z 903.73,A -85,B 0,C 180,E1 -18048.05,E2 -18048.05} C_VEL
LIN {X 0,Y 301.939,Z 915.851,A -85,B 0,C 180,E1 -18048.555,E2 -18048.555} C_VEL
LIN {X 0,Y 299.859,Z 928.217,A -85,B 0,C 180,E1 -18049.209,E2 -18049.209} C_VEL
LIN {X 0,Y 297.741,Z 939.601,A -85,B 0,C 180,E1 -18049.969,E2 -18049.969} C_VEL
LIN {X 0,Y 294.862,Z 952.834,A -85,B 0,C 180,E1 -18051.051,E2 -18051.051} C_VEL
LIN {X 0,Y 292.062,Z 964.13,A -85,B 0,C 180,E1 -18052.15,E2 -18052.15} C_VEL
LIN {X 0,Y 288.755,Z 976.236,A -85,B 0,C 180,E1 -18053.556,E2 -18053.556} C_VEL
LIN {X 0,Y 285.446,Z 987.359,A -85,B 0,C 180,E1 -18055.08,E2 -18055.08} C_VEL
LIN {X 0,Y 282.056,Z 997.853,A -85,B 0,C 180,E1 -18056.759,E2 -18056.759} C_VEL
LIN {X 0,Y 279,Z 1007.122,A -85,B 0,C 180,E1 -18058.488,E2 -18058.488} C_VEL
LIN {X 0,Y 275.603,Z 1016.975,A -85,B 0,C 180,E1 -18060.637,E2 -18060.637} C_VEL
LIN {X 0,Y 272.624,Z 1025.377,A -85,B 0,C 180,E1 -18062.77,E2 -18062.77} C_VEL
LIN {X 0,Y 269.574,Z 1033.977,A -85,B 0,C 180,E1 -18065.347,E2 -18065.347} C_VEL
LIN {X 0,Y 267.428,Z 1040.411,A -85,B 0,C 180,E1 -18067.601,E2 -18067.601} C_VEL
LIN {X 0,Y 265.031,Z 1047.676,A -85,B 0,C 180,E1 -18070.642,E2 -18070.642} C_VEL
LIN {X 0,Y 263.667,Z 1052.331,A -85,B 0,C 180,E1 -18072.951,E2 -18072.951} C_VEL
LIN {X 0,Y 262.353,Z 1057.435,A -85,B 0,C 180,E1 -18076.049,E2 -18076.049} C_VEL
LIN {X 0,Y 261.508,Z 1061.44,A -85,B 0,C 180,E1 -18079.157,E2 -18079.157} C_VEL
LIN {X 0,Y 261.137,Z 1064.404,A -85,B 0,C 180,E1 -18082.267,E2 -18082.267} C_VEL
LIN {X 0,Y 261.053,Z 1066.167,A -85,B 0,C 180,E1 -18084.941,E2 -18084.941} C_VEL
LIN {X 0,Y 261.037,Z 1067.069,A -85,B 0,C 180,E1 -18086.913,E2 -18086.913} C_VEL
LIN {X 0,Y 261.125,Z 1067.56,A -85,B 0,C 180,E1 -18090,E2 -18090} C_VEL
LIN {X 0,Y 261.037,Z 1067.069,A -85,B 0,C 180,E1 -18093.087,E2 -18093.087} C_VEL
LIN {X 0,Y 261.046,Z 1065.594,A -85,B 0,C 180,E1 -18096.182,E2 -18096.182} C_VEL
LIN {X 0,Y 261.278,Z 1063.118,A -85,B 0,C 180,E1 -18099.287,E2 -18099.287} C_VEL
LIN {X 0,Y 262.122,Z 1058.526,A -85,B 0,C 180,E1 -18103.173,E2 -18103.173} C_VEL
LIN {X 0,Y 262.951,Z 1055.031,A -85,B 0,C 180,E1 -18105.502,E2 -18105.502} C_VEL
LIN {X 0,Y 264.529,Z 1049.298,A -85,B 0,C 180,E1 -18108.591,E2 -18108.591} C_VEL
LIN {X 0,Y 266.186,Z 1044.237,A -85,B 0,C 180,E1 -18110.881,E2 -18110.881} C_VEL
LIN {X 0,Y 268.588,Z 1036.879,A -85,B 0,C 180,E1 -18113.677,E2 -18113.677} C_VEL
LIN {X 0,Y 271.264,Z 1029.216,A -85,B 0,C 180,E1 -18116.131,E2 -18116.131} C_VEL
LIN {X 0,Y 274.119,Z 1021.25,A -85,B 0,C 180,E1 -18118.314,E2 -18118.314} C_VEL
LIN {X 0,Y 277.406,Z 1011.8,A -85,B 0,C 180,E1 -18120.528,E2 -18120.528} C_VEL
LIN {X 0,Y 280.199,Z 1003.571,A -85,B 0,C 180,E1 -18122.207,E2 -18122.207} C_VEL
LIN {X 0,Y 283.953,Z 991.705,A -85,B 0,C 180,E1 -18124.268,E2 -18124.268} C_VEL
LIN {X 0,Y 287.579,Z 980.301,A -85,B 0,C 180,E1 -18125.91,E2 -18125.91} C_VEL
LIN {X 0,Y 290.529,Z 969.881,A -85,B 0,C 180,E1 -18127.21,E2 -18127.21} C_VEL
LIN {X 0,Y 293.616,Z 957.858,A -85,B 0,C 180,E1 -18128.486,E2 -18128.486} C_VEL
LIN {X 0,Y 296.503,Z 945.544,A -85,B 0,C 180,E1 -18129.568,E2 -18129.568} C_VEL
LIN {X 0,Y 298.996,Z 933.002,A -85,B 0,C 180,E1 -18130.49,E2 -18130.49} C_VEL
LIN {X 0,Y 301.303,Z 919.578,A -85,B 0,C 180,E1 -18131.273,E2 -18131.273} C_VEL
LIN {X 0,Y 303.191,Z 906.666,A -85,B 0,C 180,E1 -18131.846,E2 -18131.846} C_VEL
LIN {X 0,Y 304.64,Z 893.318,A -85,B 0,C 180,E1 -18132.289,E2 -18132.289} C_VEL
LIN {X 0,Y 306.099,Z 866.074,A -85,B 0,C 180,E1 -18132.967,E2 -18132.967} C_VEL
LIN {X 0,Y 311.199,Z 766.728,A -85,B 0,C 180,E1 -18135.198,E2 -18135.198} C_VEL
LIN {X 0,Y 302.751,Z 748.322,A -85,B 0,C 180,E1 -18137.446,E2 -18137.446} C_VEL
LIN {X 0,Y 295.384,Z 734.242,A -85,B 0,C 180,E1 -18139.527,E2 -18139.527} C_VEL
LIN {X 0,Y 289.017,Z 722.942,A -85,B 0,C 180,E1 -18141.456,E2 -18141.456} C_VEL
LIN {X 0,Y 282.058,Z 711.872,A -85,B 0,C 180,E1 -18143.714,E2 -18143.714} C_VEL
LIN {X 0,Y 279.033,Z 707.222,A -85,B 0,C 180,E1 -18144.764,E2 -18144.764} C_VEL
LIN {X 0,Y 275.148,Z 701.576,A -85,B 0,C 180,E1 -18146.174,E2 -18146.174} C_VEL
LIN {X 0,Y 271.196,Z 696.196,A -85,B 0,C 180,E1 -18147.69,E2 -18147.69} C_VEL
LIN {X 0,Y 268.703,Z 693.633,A -85,B 0,C 180,E1 -18148.662,E2 -18148.662} C_VEL
LIN {X 0,Y 267.413,Z 691.208,A -85,B 0,C 180,E1 -18149.239,E2 -18149.239} C_VEL
LIN {X 0,Y 264.866,Z 689.26,A -85,B 0,C 180,E1 -18150.273,E2 -18150.273} C_VEL
LIN {X 0,Y 263.347,Z 686.449,A -85,B 0,C 180,E1 -18151.072,E2 -18151.072} C_VEL
LIN {X 0,Y 263.217,Z 685.552,A -85,B 0,C 180,E1 -18151.603,E2 -18151.603} C_VEL
LIN {X 0,Y 263.221,Z 685.51,A -85,B 0,C 180,E1 -18155.2,E2 -18155.2} C_VEL
LIN {X 0,Y 263.259,Z 685.506,A -85,B 0,C 180,E1 -18159.693,E2 -18159.693} C_VEL
LIN {X 0,Y 263.339,Z 685.497,A -85,B 0,C 180,E1 -18164.521,E2 -18164.521} C_VEL
LIN {X 0,Y 263.368,Z 685.489,A -85,B 0,C 180,E1 -18169.234,E2 -18169.234} C_VEL
LIN {X 0,Y 263.564,Z 685.439,A -85,B 0,C 180,E1 -18172.338,E2 -18172.338} C_VEL
LIN {X 0,Y 263.745,Z 685.424,A -85,B 0,C 180,E1 -18178.473,E2 -18178.473} C_VEL
LIN {X 0,Y 263.745,Z 685.422,A -85,B 0,C 180,E1 -18181.527,E2 -18181.527} C_VEL
LIN {X 0,Y 263.563,Z 685.442,A -85,B 0,C 180,E1 -18187.661,E2 -18187.661} C_VEL
LIN {X 0,Y 263.367,Z 685.487,A -85,B 0,C 180,E1 -18190.765,E2 -18190.765} C_VEL
LIN {X 0,Y 263.338,Z 685.494,A -85,B 0,C 180,E1 -18195.478,E2 -18195.478} C_VEL
LIN {X 0,Y 263.281,Z 685.501,A -85,B 0,C 180,E1 -18200.305,E2 -18200.305} C_VEL
LIN {X 0,Y 263.204,Z 685.492,A -85,B 0,C 180,E1 -18205.291,E2 -18205.291} C_VEL
LIN {X 0,Y 263.183,Z 685.63,A -85,B 0,C 180,E1 -18208.838,E2 -18208.838} C_VEL
LIN {X 0,Y 263.484,Z 686.887,A -85,B 0,C 180,E1 -18209.458,E2 -18209.458} C_VEL
LIN {X 0,Y 265.015,Z 689.465,A -85,B 0,C 180,E1 -18210.2,E2 -18210.2} C_VEL
LIN {X 0,Y 267.511,Z 691.432,A -85,B 0,C 180,E1 -18211.215,E2 -18211.215} C_VEL
LIN {X 0,Y 269.544,Z 694.732,A -85,B 0,C 180,E1 -18212.089,E2 -18212.089} C_VEL
LIN {X 0,Y 271.886,Z 696.987,A -85,B 0,C 180,E1 -18212.982,E2 -18212.982} C_VEL
LIN {X 0,Y 274.462,Z 700.481,A -85,B 0,C 180,E1 -18213.97,E2 -18213.97} C_VEL
LIN {X 0,Y 275.978,Z 702.164,A -85,B 0,C 180,E1 -18214.514,E2 -18214.514} C_VEL
LIN {X 0,Y 279.963,Z 707.46,A -85,B 0,C 180,E1 -18215.92,E2 -18215.92} C_VEL
LIN {X 0,Y 290.769,Z 720.902,A -85,B 0,C 180,E1 -18219.301,E2 -18219.301} C_VEL
LIN {X 0,Y 297.383,Z 727.798,A -85,B 0,C 180,E1 -18221.149,E2 -18221.149} C_VEL
LIN {X 0,Y 303.204,Z 733.614,A -85,B 0,C 180,E1 -18222.843,E2 -18222.843} C_VEL
LIN {X 0,Y 306.558,Z 736.702,A -85,B 0,C 180,E1 -18223.841,E2 -18223.841} C_VEL
LIN {X 0,Y 311.167,Z 741.087,A -85,B 0,C 180,E1 -18225.325,E2 -18225.325} C_VEL
LIN {X 0,Y 317.333,Z 747.08,A -85,B 0,C 180,E1 -18227.471,E2 -18227.471} C_VEL
LIN {X 0,Y 323.558,Z 753.272,A -85,B 0,C 180,E1 -18229.846,E2 -18229.846} C_VEL
LIN {X 0,Y 326.268,Z 755.875,A -85,B 0,C 180,E1 -18230.905,E2 -18230.905} C_VEL
LIN {X 0,Y 330.367,Z 759.873,A -85,B 0,C 180,E1 -18232.547,E2 -18232.547} C_VEL
LIN {X 0,Y 332.253,Z 761.58,A -85,B 0,C 180,E1 -18233.305,E2 -18233.305} C_VEL
LIN {X 0,Y 336.95,Z 766.153,A -85,B 0,C 180,E1 -18235.284,E2 -18235.284} C_VEL
LIN {X 0,Y 339.797,Z 768.593,A -85,B 0,C 180,E1 -18236.505,E2 -18236.505} C_VEL
LIN {X 0,Y 344.236,Z 772.825,A -85,B 0,C 180,E1 -18238.495,E2 -18238.495} C_VEL
LIN {X 0,Y 347.096,Z 775.251,A -85,B 0,C 180,E1 -18239.819,E2 -18239.819} C_VEL
LIN {X 0,Y 351.021,Z 779.132,A -85,B 0,C 180,E1 -18241.756,E2 -18241.756} C_VEL
LIN {X 0,Y 354.437,Z 781.795,A -85,B 0,C 180,E1 -18243.487,E2 -18243.487} C_VEL
LIN {X 0,Y 358.064,Z 785.465,A -85,B 0,C 180,E1 -18245.489,E2 -18245.489} C_VEL
LIN {X 0,Y 361.798,Z 788.078,A -85,B 0,C 180,E1 -18247.637,E2 -18247.637} C_VEL
LIN {X 0,Y 363.821,Z 790.167,A -85,B 0,C 180,E1 -18248.934,E2 -18248.934} C_VEL
LIN {X 0,Y 367.24,Z 793.256,A -85,B 0,C 180,E1 -18251.269,E2 -18251.269} C_VEL
LIN {X 0,Y 370.223,Z 795.118,A -85,B 0,C 180,E1 -18253.457,E2 -18253.457} C_VEL
LIN {X 0,Y 371.263,Z 795.901,A -85,B 0,C 180,E1 -18254.315,E2 -18254.315} C_VEL
LIN {X 0,Y 373.492,Z 798.493,A -85,B 0,C 180,E1 -18256.41,E2 -18256.41} C_VEL
LIN {X 0,Y 375.74,Z 800.43,A -85,B 0,C 180,E1 -18258.807,E2 -18258.807} C_VEL
LIN {X 0,Y 377.504,Z 801.44,A -85,B 0,C 180,E1 -18261.028,E2 -18261.028} C_VEL
LIN {X 0,Y 379.104,Z 802.183,A -85,B 0,C 180,E1 -18263.614,E2 -18263.614} C_VEL
LIN {X 0,Y 380.231,Z 802.837,A -85,B 0,C 180,E1 -18266.465,E2 -18266.465} C_VEL
LIN {X 0,Y 380.66,Z 803.068,A -85,B 0,C 180,E1 -18268.942,E2 -18268.942} C_VEL
LIN {X 0,Y 380.66,Z 803.07,A -85,B 0,C 180,E1 -18271.058,E2 -18271.058} C_VEL
LIN {X 0,Y 380.231,Z 802.837,A -85,B 0,C 180,E1 -18273.535,E2 -18273.535} C_VEL
LIN {X 0,Y 379.109,Z 802.139,A -85,B 0,C 180,E1 -18276.386,E2 -18276.386} C_VEL
LIN {X 0,Y 377.806,Z 801.58,A -85,B 0,C 180,E1 -18278.558,E2 -18278.558} C_VEL
LIN {X 0,Y 375.832,Z 800.492,A -85,B 0,C 180,E1 -18281.082,E2 -18281.082} C_VEL
LIN {X 0,Y 373.491,Z 798.493,A -85,B 0,C 180,E1 -18283.59,E2 -18283.59} C_VEL
LIN {X 0,Y 371.066,Z 795.63,A -85,B 0,C 180,E1 -18285.864,E2 -18285.864} C_VEL
LIN {X 0,Y 367.667,Z 793.578,A -85,B 0,C 180,E1 -18288.427,E2 -18288.427} C_VEL
LIN {X 0,Y 364.265,Z 790.604,A -85,B 0,C 180,E1 -18290.787,E2 -18290.787} C_VEL
LIN {X 0,Y 361.8,Z 788.055,A -85,B 0,C 180,E1 -18292.364,E2 -18292.364} C_VEL
LIN {X 0,Y 357.946,Z 785.348,A -85,B 0,C 180,E1 -18294.581,E2 -18294.581} C_VEL
LIN {X 0,Y 354.057,Z 781.377,A -85,B 0,C 180,E1 -18296.718,E2 -18296.718} C_VEL
LIN {X 0,Y 349.546,Z 777.801,A -85,B 0,C 180,E1 -18298.977,E2 -18298.977} C_VEL
LIN {X 0,Y 345.631,Z 773.863,A -85,B 0,C 180,E1 -18300.864,E2 -18300.864} C_VEL
LIN {X 0,Y 341.253,Z 770.122,A -85,B 0,C 180,E1 -18302.849,E2 -18302.849} C_VEL
LIN {X 0,Y 338.08,Z 767.003,A -85,B 0,C 180,E1 -18304.246,E2 -18304.246} C_VEL
LIN {X 0,Y 333.517,Z 762.966,A -85,B 0,C 180,E1 -18306.158,E2 -18306.158} C_VEL
LIN {X 0,Y 330.805,Z 760.224,A -85,B 0,C 180,E1 -18307.281,E2 -18307.281} C_VEL
LIN {X 0,Y 326.167,Z 755.833,A -85,B 0,C 180,E1 -18309.132,E2 -18309.132} C_VEL
LIN {X 0,Y 323.405,Z 753.148,A -85,B 0,C 180,E1 -18310.212,E2 -18310.212} C_VEL
LIN {X 0,Y 318.764,Z 748.33,A -85,B 0,C 180,E1 -18312.002,E2 -18312.002} C_VEL
LIN {X 0,Y 313.607,Z 743.516,A -85,B 0,C 180,E1 -18313.846,E2 -18313.846} C_VEL
LIN {X 0,Y 311.162,Z 741.058,A -85,B 0,C 180,E1 -18314.678,E2 -18314.678} C_VEL
LIN {X 0,Y 306.556,Z 736.689,A -85,B 0,C 180,E1 -18316.16,E2 -18316.16} C_VEL
LIN {X 0,Y 299.954,Z 730.367,A -85,B 0,C 180,E1 -18318.126,E2 -18318.126} C_VEL
LIN {X 0,Y 293.279,Z 723.551,A -85,B 0,C 180,E1 -18320,E2 -18320} C_VEL
LIN {X 0,Y 287.251,Z 716.742,A -85,B 0,C 180,E1 -18321.735,E2 -18321.735} C_VEL
LIN {X 0,Y 282.855,Z 711.106,A -85,B 0,C 180,E1 -18323.121,E2 -18323.121} C_VEL
LIN {X 0,Y 279.223,Z 706.289,A -85,B 0,C 180,E1 -18324.343,E2 -18324.343} C_VEL
LIN {X 0,Y 275.873,Z 701.979,A -85,B 0,C 180,E1 -18325.527,E2 -18325.527} C_VEL
LIN {X 0,Y 272.277,Z 697.676,A -85,B 0,C 180,E1 -18326.857,E2 -18326.857} C_VEL
LIN {X 0,Y 271.262,Z 696.224,A -85,B 0,C 180,E1 -18327.26,E2 -18327.26} C_VEL
LIN {X 0,Y 268.729,Z 693.682,A -85,B 0,C 180,E1 -18328.243,E2 -18328.243} C_VEL
LIN {X 0,Y 267.382,Z 691.181,A -85,B 0,C 180,E1 -18328.844,E2 -18328.844} C_VEL
LIN {X 0,Y 264.726,Z 689.09,A -85,B 0,C 180,E1 -18329.928,E2 -18329.928} C_VEL
LIN {X 0,Y 263.308,Z 686.277,A -85,B 0,C 180,E1 -18330.74,E2 -18330.74} C_VEL
LIN {X 0,Y 263.176,Z 685.518,A -85,B 0,C 180,E1 -18331.271,E2 -18331.271} C_VEL
LIN {X 0,Y 263.222,Z 685.508,A -85,B 0,C 180,E1 -18335.199,E2 -18335.199} C_VEL
LIN {X 0,Y 263.281,Z 685.501,A -85,B 0,C 180,E1 -18339.695,E2 -18339.695} C_VEL
LIN {X 0,Y 263.338,Z 685.493,A -85,B 0,C 180,E1 -18344.522,E2 -18344.522} C_VEL
LIN {X 0,Y 263.367,Z 685.484,A -85,B 0,C 180,E1 -18349.235,E2 -18349.235} C_VEL
LIN {X 0,Y 263.561,Z 685.44,A -85,B 0,C 180,E1 -18352.339,E2 -18352.339} C_VEL
LIN {X 0,Y 263.745,Z 685.423,A -85,B 0,C 180,E1 -18358.473,E2 -18358.473} C_VEL
LIN {X 0,Y 263.745,Z 685.426,A -85,B 0,C 180,E1 -18361.527,E2 -18361.527} C_VEL
LIN {X 0,Y 263.564,Z 685.439,A -85,B 0,C 180,E1 -18367.662,E2 -18367.662} C_VEL
LIN {X 0,Y 263.368,Z 685.487,A -85,B 0,C 180,E1 -18370.766,E2 -18370.766} C_VEL
LIN {X 0,Y 263.339,Z 685.494,A -85,B 0,C 180,E1 -18375.479,E2 -18375.479} C_VEL
LIN {X 0,Y 263.259,Z 685.506,A -85,B 0,C 180,E1 -18380.307,E2 -18380.307} C_VEL
LIN {X 0,Y 263.203,Z 685.495,A -85,B 0,C 180,E1 -18385.292,E2 -18385.292} C_VEL
LIN {X 0,Y 263.22,Z 685.693,A -85,B 0,C 180,E1 -18388.56,E2 -18388.56} C_VEL
LIN {X 0,Y 263.527,Z 686.952,A -85,B 0,C 180,E1 -18389.07,E2 -18389.07} C_VEL
LIN {X 0,Y 265.061,Z 689.493,A -85,B 0,C 180,E1 -18389.812,E2 -18389.812} C_VEL
LIN {X 0,Y 267.521,Z 691.502,A -85,B 0,C 180,E1 -18390.815,E2 -18390.815} C_VEL
LIN {X 0,Y 269.485,Z 694.652,A -85,B 0,C 180,E1 -18391.658,E2 -18391.658} C_VEL
LIN {X 0,Y 271.834,Z 696.897,A -85,B 0,C 180,E1 -18392.554,E2 -18392.554} C_VEL
LIN {X 0,Y 276.895,Z 704.024,A -85,B 0,C 180,E1 -18394.467,E2 -18394.467} C_VEL
LIN {X 0,Y 278.394,Z 706.366,A -85,B 0,C 180,E1 -18395.013,E2 -18395.013} C_VEL
LIN {X 0,Y 280.539,Z 710.295,A -85,B 0,C 180,E1 -18395.797,E2 -18395.797} C_VEL
LIN {X 0,Y 282.16,Z 715.036,A -85,B 0,C 180,E1 -18396.446,E2 -18396.446} C_VEL
LIN {X 0,Y 284.911,Z 725.272,A -85,B 0,C 180,E1 -18397.598,E2 -18397.598} C_VEL
LIN {X 0,Y 286.669,Z 730.043,A -85,B 0,C 180,E1 -18398.237,E2 -18398.237} C_VEL
LIN {X 0,Y 287.392,Z 731.48,A -85,B 0,C 180,E1 -18398.474,E2 -18398.474} C_VEL
LIN {X 0,Y 293.707,Z 743.083,A -85,B 0,C 180,E1 -18400.417,E2 -18400.417} C_VEL
LIN {X 0,Y 300.546,Z 756.872,A -85,B 0,C 180,E1 -18402.394,E2 -18402.394} C_VEL
LIN {X 0,Y 306.133,Z 769.384,A -85,B 0,C 180,E1 -18403.934,E2 -18403.934} C_VEL
LIN {X 0,Y 299.626,Z 889.594,A -85,B 0,C 180,E1 -18406.684,E2 -18406.684} C_VEL
LIN {X 0,Y 298.434,Z 902.546,A -85,B 0,C 180,E1 -18407.101,E2 -18407.101} C_VEL
LIN {X 0,Y 296.649,Z 915.646,A -85,B 0,C 180,E1 -18407.646,E2 -18407.646} C_VEL
LIN {X 0,Y 294.505,Z 928.011,A -85,B 0,C 180,E1 -18408.304,E2 -18408.304} C_VEL
LIN {X 0,Y 292.308,Z 939.395,A -85,B 0,C 180,E1 -18409.068,E2 -18409.068} C_VEL
LIN {X 0,Y 289.348,Z 952.628,A -85,B 0,C 180,E1 -18410.163,E2 -18410.163} C_VEL
LIN {X 0,Y 286.444,Z 963.923,A -85,B 0,C 180,E1 -18411.271,E2 -18411.271} C_VEL
LIN {X 0,Y 282.768,Z 976.883,A -85,B 0,C 180,E1 -18412.808,E2 -18412.808} C_VEL
LIN {X 0,Y 279.235,Z 988.239,A -85,B 0,C 180,E1 -18414.408,E2 -18414.408} C_VEL
LIN {X 0,Y 276.073,Z 997.645,A -85,B 0,C 180,E1 -18415.941,E2 -18415.941} C_VEL
LIN {X 0,Y 272.887,Z 1006.914,A -85,B 0,C 180,E1 -18417.698,E2 -18417.698} C_VEL
LIN {X 0,Y 269.289,Z 1016.926,A -85,B 0,C 180,E1 -18419.925,E2 -18419.925} C_VEL
LIN {X 0,Y 266.196,Z 1025.167,A -85,B 0,C 180,E1 -18422.056,E2 -18422.056} C_VEL
LIN {X 0,Y 263.013,Z 1033.768,A -85,B 0,C 180,E1 -18424.689,E2 -18424.689} C_VEL
LIN {X 0,Y 260.769,Z 1040.203,A -85,B 0,C 180,E1 -18426.997,E2 -18426.997} C_VEL
LIN {X 0,Y 258.248,Z 1047.467,A -85,B 0,C 180,E1 -18430.113,E2 -18430.113} C_VEL
LIN {X 0,Y 256.78,Z 1052.122,A -85,B 0,C 180,E1 -18432.479,E2 -18432.479} C_VEL
LIN {X 0,Y 255.385,Z 1057.227,A -85,B 0,C 180,E1 -18435.661,E2 -18435.661} C_VEL
LIN {X 0,Y 254.463,Z 1061.233,A -85,B 0,C 180,E1 -18438.853,E2 -18438.853} C_VEL
LIN {X 0,Y 254.067,Z 1064.198,A -85,B 0,C 180,E1 -18442.05,E2 -18442.05} C_VEL
LIN {X 0,Y 253.945,Z 1066.085,A -85,B 0,C 180,E1 -18445.077,E2 -18445.077} C_VEL
LIN {X 0,Y 253.935,Z 1066.863,A -85,B 0,C 180,E1 -18446.827,E2 -18446.827} C_VEL
LIN {X 0,Y 254.053,Z 1067.356,A -85,B 0,C 180,E1 -18450,E2 -18450} C_VEL
LIN {X 0,Y 253.935,Z 1066.863,A -85,B 0,C 180,E1 -18453.173,E2 -18453.173} C_VEL
LIN {X 0,Y 253.956,Z 1065.388,A -85,B 0,C 180,E1 -18456.355,E2 -18456.355} C_VEL
LIN {X 0,Y 254.221,Z 1062.911,A -85,B 0,C 180,E1 -18459.548,E2 -18459.548} C_VEL
LIN {X 0,Y 255.133,Z 1058.318,A -85,B 0,C 180,E1 -18463.541,E2 -18463.541} C_VEL
LIN {X 0,Y 256.107,Z 1054.427,A -85,B 0,C 180,E1 -18466.166,E2 -18466.166} C_VEL
LIN {X 0,Y 257.719,Z 1049.09,A -85,B 0,C 180,E1 -18469.101,E2 -18469.101} C_VEL
LIN {X 0,Y 259.461,Z 1044.028,A -85,B 0,C 180,E1 -18471.448,E2 -18471.448} C_VEL
LIN {X 0,Y 262.265,Z 1035.892,A -85,B 0,C 180,E1 -18474.579,E2 -18474.579} C_VEL
LIN {X 0,Y 264.82,Z 1029.008,A -85,B 0,C 180,E1 -18476.817,E2 -18476.817} C_VEL
LIN {X 0,Y 267.829,Z 1021.042,A -85,B 0,C 180,E1 -18479.041,E2 -18479.041} C_VEL
LIN {X 0,Y 271.11,Z 1011.93,A -85,B 0,C 180,E1 -18481.228,E2 -18481.228} C_VEL
LIN {X 0,Y 274.153,Z 1003.363,A -85,B 0,C 180,E1 -18483.007,E2 -18483.007} C_VEL
LIN {X 0,Y 278.066,Z 991.498,A -85,B 0,C 180,E1 -18485.098,E2 -18485.098} C_VEL
LIN {X 0,Y 281.83,Z 980.095,A -85,B 0,C 180,E1 -18486.761,E2 -18486.761} C_VEL
LIN {X 0,Y 284.881,Z 969.675,A -85,B 0,C 180,E1 -18488.078,E2 -18488.078} C_VEL
LIN {X 0,Y 288.062,Z 957.652,A -85,B 0,C 180,E1 -18489.369,E2 -18489.369} C_VEL
LIN {X 0,Y 291.042,Z 945.338,A -85,B 0,C 180,E1 -18490.463,E2 -18490.463} C_VEL
LIN {X 0,Y 293.623,Z 932.796,A -85,B 0,C 180,E1 -18491.391,E2 -18491.391} C_VEL
LIN {X 0,Y 296.019,Z 919.373,A -85,B 0,C 180,E1 -18492.177,E2 -18492.177} C_VEL
LIN {X 0,Y 297.945,Z 906.461,A -85,B 0,C 180,E1 -18492.756,E2 -18492.756} C_VEL
LIN {X 0,Y 299.445,Z 892.738,A -85,B 0,C 180,E1 -18493.216,E2 -18493.216} C_VEL
LIN {X 0,Y 301.003,Z 864.768,A -85,B 0,C 180,E1 -18493.913,E2 -18493.913} C_VEL
LIN {X 0,Y 306.109,Z 769.241,A -85,B 0,C 180,E1 -18496.076,E2 -18496.076} C_VEL
LIN {X 0,Y 298.245,Z 751.983,A -85,B 0,C 180,E1 -18498.261,E2 -18498.261} C_VEL
LIN {X 0,Y 291.219,Z 738.409,A -85,B 0,C 180,E1 -18500.333,E2 -18500.333} C_VEL
LIN {X 0,Y 285.23,Z 727.659,A -85,B 0,C 180,E1 -18502.224,E2 -18502.224} C_VEL
LIN {X 0,Y 278.801,Z 717.229,A -85,B 0,C 180,E1 -18504.397,E2 -18504.397} C_VEL
LIN {X 0,Y 275.509,Z 712.171,A -85,B 0,C 180,E1 -18505.584,E2 -18505.584} C_VEL
LIN {X 0,Y 272.21,Z 707.243,A -85,B 0,C 180,E1 -18506.834,E2 -18506.834} C_VEL
LIN {X 0,Y 268.571,Z 702.289,A -85,B 0,C 180,E1 -18508.277,E2 -18508.277} C_VEL
LIN {X 0,Y 265.932,Z 699.321,A -85,B 0,C 180,E1 -18509.354,E2 -18509.354} C_VEL
LIN {X 0,Y 264.663,Z 697.373,A -85,B 0,C 180,E1 -18509.919,E2 -18509.919} C_VEL
LIN {X 0,Y 262.095,Z 694.907,A -85,B 0,C 180,E1 -18511.03,E2 -18511.03} C_VEL
LIN {X 0,Y 260.337,Z 691.99,A -85,B 0,C 180,E1 -18511.897,E2 -18511.897} C_VEL
LIN {X 0,Y 257.846,Z 690.112,A -85,B 0,C 180,E1 -18513.054,E2 -18513.054} C_VEL
LIN {X 0,Y 256.423,Z 687.618,A -85,B 0,C 180,E1 -18513.881,E2 -18513.881} C_VEL
LIN {X 0,Y 256.174,Z 686.5,A -85,B 0,C 180,E1 -18514.567,E2 -18514.567} C_VEL
LIN {X 0,Y 256.162,Z 686.38,A -85,B 0,C 180,E1 -18519.104,E2 -18519.104} C_VEL
LIN {X 0,Y 256.274,Z 686.371,A -85,B 0,C 180,E1 -18524.083,E2 -18524.083} C_VEL
LIN {X 0,Y 256.304,Z 686.363,A -85,B 0,C 180,E1 -18528.933,E2 -18528.933} C_VEL
LIN {X 0,Y 256.532,Z 686.314,A -85,B 0,C 180,E1 -18532.126,E2 -18532.126} C_VEL
LIN {X 0,Y 256.708,Z 686.3,A -85,B 0,C 180,E1 -18538.431,E2 -18538.431} C_VEL
LIN {X 0,Y 256.708,Z 686.297,A -85,B 0,C 180,E1 -18541.568,E2 -18541.568} C_VEL
LIN {X 0,Y 256.531,Z 686.317,A -85,B 0,C 180,E1 -18547.873,E2 -18547.873} C_VEL
LIN {X 0,Y 256.302,Z 686.36,A -85,B 0,C 180,E1 -18551.066,E2 -18551.066} C_VEL
LIN {X 0,Y 256.288,Z 686.364,A -85,B 0,C 180,E1 -18555.915,E2 -18555.915} C_VEL
LIN {X 0,Y 256.226,Z 686.369,A -85,B 0,C 180,E1 -18560.889,E2 -18560.889} C_VEL
LIN {X 0,Y 256.155,Z 686.427,A -85,B 0,C 180,E1 -18565.77,E2 -18565.77} C_VEL
LIN {X 0,Y 256.361,Z 687.423,A -85,B 0,C 180,E1 -18566.454,E2 -18566.454} C_VEL
LIN {X 0,Y 257.983,Z 690.295,A -85,B 0,C 180,E1 -18567.423,E2 -18567.423} C_VEL
LIN {X 0,Y 260.749,Z 692.496,A -85,B 0,C 180,E1 -18568.707,E2 -18568.707} C_VEL
LIN {X 0,Y 262.624,Z 695.573,A -85,B 0,C 180,E1 -18569.619,E2 -18569.619} C_VEL
LIN {X 0,Y 265.056,Z 697.782,A -85,B 0,C 180,E1 -18570.654,E2 -18570.654} C_VEL
LIN {X 0,Y 267.473,Z 701.314,A -85,B 0,C 180,E1 -18571.702,E2 -18571.702} C_VEL
LIN {X 0,Y 269.359,Z 703.246,A -85,B 0,C 180,E1 -18572.445,E2 -18572.445} C_VEL
LIN {X 0,Y 272.276,Z 706.972,A -85,B 0,C 180,E1 -18573.581,E2 -18573.581} C_VEL
LIN {X 0,Y 277.102,Z 713.371,A -85,B 0,C 180,E1 -18575.35,E2 -18575.35} C_VEL
LIN {X 0,Y 288.154,Z 727.213,A -85,B 0,C 180,E1 -18578.904,E2 -18578.904} C_VEL
LIN {X 0,Y 294.864,Z 734.152,A -85,B 0,C 180,E1 -18580.777,E2 -18580.777} C_VEL
LIN {X 0,Y 300.964,Z 740.134,A -85,B 0,C 180,E1 -18582.511,E2 -18582.511} C_VEL
LIN {X 0,Y 304.753,Z 743.726,A -85,B 0,C 180,E1 -18583.649,E2 -18583.649} C_VEL
LIN {X 0,Y 311.135,Z 749.65,A -85,B 0,C 180,E1 -18585.69,E2 -18585.69} C_VEL
LIN {X 0,Y 315.866,Z 754.085,A -85,B 0,C 180,E1 -18587.326,E2 -18587.326} C_VEL
LIN {X 0,Y 321.454,Z 759.682,A -85,B 0,C 180,E1 -18589.43,E2 -18589.43} C_VEL
LIN {X 0,Y 324.323,Z 762.415,A -85,B 0,C 180,E1 -18590.535,E2 -18590.535} C_VEL
LIN {X 0,Y 328.936,Z 766.778,A -85,B 0,C 180,E1 -18592.371,E2 -18592.371} C_VEL
LIN {X 0,Y 335.05,Z 772.625,A -85,B 0,C 180,E1 -18594.89,E2 -18594.89} C_VEL
LIN {X 0,Y 338.305,Z 775.467,A -85,B 0,C 180,E1 -18596.278,E2 -18596.278} C_VEL
LIN {X 0,Y 342.83,Z 779.685,A -85,B 0,C 180,E1 -18598.3,E2 -18598.3} C_VEL
LIN {X 0,Y 345.746,Z 782.236,A -85,B 0,C 180,E1 -18599.644,E2 -18599.644} C_VEL
LIN {X 0,Y 349.839,Z 786.099,A -85,B 0,C 180,E1 -18601.633,E2 -18601.633} C_VEL
LIN {X 0,Y 353.094,Z 788.66,A -85,B 0,C 180,E1 -18603.274,E2 -18603.274} C_VEL
LIN {X 0,Y 356.766,Z 792.311,A -85,B 0,C 180,E1 -18605.27,E2 -18605.27} C_VEL
LIN {X 0,Y 360.774,Z 795.103,A -85,B 0,C 180,E1 -18607.57,E2 -18607.57} C_VEL
LIN {X 0,Y 364.217,Z 798.621,A -85,B 0,C 180,E1 -18609.807,E2 -18609.807} C_VEL
LIN {X 0,Y 367.649,Z 801.258,A -85,B 0,C 180,E1 -18612.191,E2 -18612.191} C_VEL
LIN {X 0,Y 370.215,Z 802.86,A -85,B 0,C 180,E1 -18614.176,E2 -18614.176} C_VEL
LIN {X 0,Y 372.573,Z 805.568,A -85,B 0,C 180,E1 -18616.375,E2 -18616.375} C_VEL
LIN {X 0,Y 374.674,Z 807.345,A -85,B 0,C 180,E1 -18618.567,E2 -18618.567} C_VEL
LIN {X 0,Y 376.445,Z 808.42,A -85,B 0,C 180,E1 -18620.778,E2 -18620.778} C_VEL
LIN {X 0,Y 377.902,Z 809.159,A -85,B 0,C 180,E1 -18623.026,E2 -18623.026} C_VEL
LIN {X 0,Y 378.964,Z 809.668,A -85,B 0,C 180,E1 -18625.296,E2 -18625.296} C_VEL
LIN {X 0,Y 379.679,Z 810.028,A -85,B 0,C 180,E1 -18627.878,E2 -18627.878} C_VEL
LIN {X 0,Y 379.878,Z 810.099,A -85,B 0,C 180,E1 -18630,E2 -18630} C_VEL
LIN {X 0,Y 379.679,Z 810.028,A -85,B 0,C 180,E1 -18632.122,E2 -18632.122} C_VEL
LIN {X 0,Y 378.964,Z 809.666,A -85,B 0,C 180,E1 -18634.704,E2 -18634.704} C_VEL
LIN {X 0,Y 377.714,Z 809.038,A -85,B 0,C 180,E1 -18637.302,E2 -18637.302} C_VEL
LIN {X 0,Y 375.794,Z 808.074,A -85,B 0,C 180,E1 -18640.107,E2 -18640.107} C_VEL
LIN {X 0,Y 373.553,Z 806.468,A -85,B 0,C 180,E1 -18642.626,E2 -18642.626} C_VEL
LIN {X 0,Y 371.106,Z 803.975,A -85,B 0,C 180,E1 -18645.022,E2 -18645.022} C_VEL
LIN {X 0,Y 369.631,Z 802.317,A -85,B 0,C 180,E1 -18646.309,E2 -18646.309} C_VEL
LIN {X 0,Y 366.488,Z 800.459,A -85,B 0,C 180,E1 -18648.63,E2 -18648.63} C_VEL
LIN {X 0,Y 362.922,Z 797.375,A -85,B 0,C 180,E1 -18651.055,E2 -18651.055} C_VEL
LIN {X 0,Y 360.536,Z 794.932,A -85,B 0,C 180,E1 -18652.57,E2 -18652.57} C_VEL
LIN {X 0,Y 356.434,Z 792.038,A -85,B 0,C 180,E1 -18654.907,E2 -18654.907} C_VEL
LIN {X 0,Y 351.815,Z 787.537,A -85,B 0,C 180,E1 -18657.398,E2 -18657.398} C_VEL
LIN {X 0,Y 347.586,Z 784.129,A -85,B 0,C 180,E1 -18659.465,E2 -18659.465} C_VEL
LIN {X 0,Y 343.982,Z 780.552,A -85,B 0,C 180,E1 -18661.189,E2 -18661.189} C_VEL
LIN {X 0,Y 339.333,Z 776.53,A -85,B 0,C 180,E1 -18663.261,E2 -18663.261} C_VEL
LIN {X 0,Y 336.341,Z 773.627,A -85,B 0,C 180,E1 -18664.566,E2 -18664.566} C_VEL
LIN {X 0,Y 331.698,Z 769.53,A -85,B 0,C 180,E1 -18666.502,E2 -18666.502} C_VEL
LIN {X 0,Y 328.898,Z 766.766,A -85,B 0,C 180,E1 -18667.643,E2 -18667.643} C_VEL
LIN {X 0,Y 324.054,Z 762.135,A -85,B 0,C 180,E1 -18669.572,E2 -18669.572} C_VEL
LIN {X 0,Y 321.076,Z 759.323,A -85,B 0,C 180,E1 -18670.718,E2 -18670.718} C_VEL
LIN {X 0,Y 315.277,Z 753.61,A -85,B 0,C 180,E1 -18672.873,E2 -18672.873} C_VEL
LIN {X 0,Y 310.823,Z 749.289,A -85,B 0,C 180,E1 -18674.42,E2 -18674.42} C_VEL
LIN {X 0,Y 304.616,Z 743.568,A -85,B 0,C 180,E1 -18676.391,E2 -18676.391} C_VEL
LIN {X 0,Y 299.739,Z 739.05,A -85,B 0,C 180,E1 -18677.843,E2 -18677.843} C_VEL
LIN {X 0,Y 293.334,Z 732.739,A -85,B 0,C 180,E1 -18679.641,E2 -18679.641} C_VEL
LIN {X 0,Y 284.468,Z 722.909,A -85,B 0,C 180,E1 -18682.206,E2 -18682.206} C_VEL
LIN {X 0,Y 275.003,Z 710.582,A -85,B 0,C 180,E1 -18685.402,E2 -18685.402} C_VEL
LIN {X 0,Y 272.113,Z 706.805,A -85,B 0,C 180,E1 -18686.479,E2 -18686.479} C_VEL
LIN {X 0,Y 269.26,Z 703.07,A -85,B 0,C 180,E1 -18687.597,E2 -18687.597} C_VEL
LIN {X 0,Y 265.951,Z 699.36,A -85,B 0,C 180,E1 -18688.938,E2 -18688.938} C_VEL
LIN {X 0,Y 264.923,Z 697.504,A -85,B 0,C 180,E1 -18689.409,E2 -18689.409} C_VEL
LIN {X 0,Y 262.243,Z 695.104,A -85,B 0,C 180,E1 -18690.555,E2 -18690.555} C_VEL
LIN {X 0,Y 260.335,Z 691.977,A -85,B 0,C 180,E1 -18691.491,E2 -18691.491} C_VEL
LIN {X 0,Y 257.718,Z 689.964,A -85,B 0,C 180,E1 -18692.712,E2 -18692.712} C_VEL
LIN {X 0,Y 256.288,Z 687.174,A -85,B 0,C 180,E1 -18693.648,E2 -18693.648} C_VEL
LIN {X 0,Y 256.155,Z 686.436,A -85,B 0,C 180,E1 -18694.23,E2 -18694.23} C_VEL
LIN {X 0,Y 256.226,Z 686.37,A -85,B 0,C 180,E1 -18699.111,E2 -18699.111} C_VEL
LIN {X 0,Y 256.288,Z 686.363,A -85,B 0,C 180,E1 -18704.085,E2 -18704.085} C_VEL
LIN {X 0,Y 256.302,Z 686.358,A -85,B 0,C 180,E1 -18708.934,E2 -18708.934} C_VEL
LIN {X 0,Y 256.529,Z 686.315,A -85,B 0,C 180,E1 -18712.127,E2 -18712.127} C_VEL
LIN {X 0,Y 256.708,Z 686.298,A -85,B 0,C 180,E1 -18718.432,E2 -18718.432} C_VEL
LIN {X 0,Y 256.708,Z 686.301,A -85,B 0,C 180,E1 -18721.569,E2 -18721.569} C_VEL
LIN {X 0,Y 256.532,Z 686.314,A -85,B 0,C 180,E1 -18727.874,E2 -18727.874} C_VEL
LIN {X 0,Y 256.304,Z 686.361,A -85,B 0,C 180,E1 -18731.067,E2 -18731.067} C_VEL
LIN {X 0,Y 256.274,Z 686.368,A -85,B 0,C 180,E1 -18735.917,E2 -18735.917} C_VEL
LIN {X 0,Y 256.162,Z 686.379,A -85,B 0,C 180,E1 -18740.896,E2 -18740.896} C_VEL
LIN {X 0,Y 256.179,Z 686.526,A -85,B 0,C 180,E1 -18745.5,E2 -18745.5} C_VEL
LIN {X 0,Y 256.461,Z 687.778,A -85,B 0,C 180,E1 -18746.17,E2 -18746.17} C_VEL
LIN {X 0,Y 257.844,Z 690.134,A -85,B 0,C 180,E1 -18746.946,E2 -18746.946} C_VEL
LIN {X 0,Y 260.331,Z 691.985,A -85,B 0,C 180,E1 -18748.1,E2 -18748.1} C_VEL
LIN {X 0,Y 260.955,Z 692.939,A -85,B 0,C 180,E1 -18748.407,E2 -18748.407} C_VEL
LIN {X 0,Y 262.856,Z 695.843,A -85,B 0,C 180,E1 -18749.316,E2 -18749.316} C_VEL
LIN {X 0,Y 265.132,Z 697.947,A -85,B 0,C 180,E1 -18750.284,E2 -18750.284} C_VEL
LIN {X 0,Y 267.541,Z 701.375,A -85,B 0,C 180,E1 -18751.322,E2 -18751.322} C_VEL
LIN {X 0,Y 269.397,Z 703.322,A -85,B 0,C 180,E1 -18752.055,E2 -18752.055} C_VEL
LIN {X 0,Y 274.028,Z 709.905,A -85,B 0,C 180,E1 -18753.861,E2 -18753.861} C_VEL
LIN {X 0,Y 277.917,Z 715.815,A -85,B 0,C 180,E1 -18755.287,E2 -18755.287} C_VEL
LIN {X 0,Y 283.828,Z 725.342,A -85,B 0,C 180,E1 -18757.318,E2 -18757.318} C_VEL
LIN {X 0,Y 287.392,Z 731.48,A -85,B 0,C 180,E1 -18758.474,E2 -18758.474} C_VEL
LIN {X 0,Y 289.31,Z 736.015,A -85,B 0,C 180,E1 -18759.121,E2 -18759.121} C_VEL
LIN {X 0,Y 291.473,Z 744.686,A -85,B 0,C 180,E1 -18759.963,E2 -18759.963} C_VEL
LIN {X 0,Y 293.975,Z 755.331,A -85,B 0,C 180,E1 -18760.926,E2 -18760.926} C_VEL
LIN {X 0,Y 295.175,Z 758.578,A -85,B 0,C 180,E1 -18761.309,E2 -18761.309} C_VEL
LIN {X 0,Y 301.074,Z 771.847,A -85,B 0,C 180,E1 -18763.016,E2 -18763.016} C_VEL
LIN {X 0,Y 294.421,Z 890.456,A -85,B 0,C 180,E1 -18765.769,E2 -18765.769} C_VEL
LIN {X 0,Y 293.148,Z 903.319,A -85,B 0,C 180,E1 -18766.193,E2 -18766.193} C_VEL
LIN {X 0,Y 291.445,Z 915.44,A -85,B 0,C 180,E1 -18766.707,E2 -18766.707} C_VEL
LIN {X 0,Y 289.22,Z 927.805,A -85,B 0,C 180,E1 -18767.364,E2 -18767.364} C_VEL
LIN {X 0,Y 286.973,Z 939.189,A -85,B 0,C 180,E1 -18768.138,E2 -18768.138} C_VEL
LIN {X 0,Y 283.901,Z 952.421,A -85,B 0,C 180,E1 -18769.24,E2 -18769.24} C_VEL
LIN {X 0,Y 280.897,Z 963.716,A -85,B 0,C 180,E1 -18770.358,E2 -18770.358} C_VEL
LIN {X 0,Y 277.073,Z 976.675,A -85,B 0,C 180,E1 -18771.909,E2 -18771.909} C_VEL
LIN {X 0,Y 273.783,Z 986.943,A -85,B 0,C 180,E1 -18773.358,E2 -18773.358} C_VEL
LIN {X 0,Y 270.142,Z 997.437,A -85,B 0,C 180,E1 -18775.087,E2 -18775.087} C_VEL
LIN {X 0,Y 266.836,Z 1006.706,A -85,B 0,C 180,E1 -18776.872,E2 -18776.872} C_VEL
LIN {X 0,Y 263.056,Z 1016.779,A -85,B 0,C 180,E1 -18779.154,E2 -18779.154} C_VEL
LIN {X 0,Y 259.357,Z 1026.239,A -85,B 0,C 180,E1 -18781.693,E2 -18781.693} C_VEL
LIN {X 0,Y 256.527,Z 1033.56,A -85,B 0,C 180,E1 -18784.002,E2 -18784.002} C_VEL
LIN {X 0,Y 254.14,Z 1039.994,A -85,B 0,C 180,E1 -18786.361,E2 -18786.361} C_VEL
LIN {X 0,Y 251.47,Z 1047.258,A -85,B 0,C 180,E1 -18789.553,E2 -18789.553} C_VEL
LIN {X 0,Y 249.903,Z 1051.913,A -85,B 0,C 180,E1 -18791.98,E2 -18791.98} C_VEL
LIN {X 0,Y 248.434,Z 1057.019,A -85,B 0,C 180,E1 -18795.25,E2 -18795.25} C_VEL
LIN {X 0,Y 247.424,Z 1061.025,A -85,B 0,C 180,E1 -18798.532,E2 -18798.532} C_VEL
LIN {X 0,Y 246.989,Z 1063.991,A -85,B 0,C 180,E1 -18801.821,E2 -18801.821} C_VEL
LIN {X 0,Y 246.87,Z 1065.181,A -85,B 0,C 180,E1 -18803.462,E2 -18803.462} C_VEL
LIN {X 0,Y 246.837,Z 1066.657,A -85,B 0,C 180,E1 -18806.736,E2 -18806.736} C_VEL
LIN {X 0,Y 246.982,Z 1067.151,A -85,B 0,C 180,E1 -18810,E2 -18810} C_VEL
LIN {X 0,Y 246.837,Z 1066.657,A -85,B 0,C 180,E1 -18813.264,E2 -18813.264} C_VEL
LIN {X 0,Y 246.87,Z 1065.181,A -85,B 0,C 180,E1 -18816.538,E2 -18816.538} C_VEL
LIN {X 0,Y 247.16,Z 1062.704,A -85,B 0,C 180,E1 -18819.823,E2 -18819.823} C_VEL
LIN {X 0,Y 248.162,Z 1058.11,A -85,B 0,C 180,E1 -18823.929,E2 -18823.929} C_VEL
LIN {X 0,Y 249.118,Z 1054.553,A -85,B 0,C 180,E1 -18826.424,E2 -18826.424} C_VEL
LIN {X 0,Y 250.908,Z 1048.881,A -85,B 0,C 180,E1 -18829.64,E2 -18829.64} C_VEL
LIN {X 0,Y 252.773,Z 1043.82,A -85,B 0,C 180,E1 -18832.045,E2 -18832.045} C_VEL
LIN {X 0,Y 255.683,Z 1035.785,A -85,B 0,C 180,E1 -18835.216,E2 -18835.216} C_VEL
LIN {X 0,Y 258.403,Z 1028.799,A -85,B 0,C 180,E1 -18837.539,E2 -18837.539} C_VEL
LIN {X 0,Y 261.571,Z 1020.835,A -85,B 0,C 180,E1 -18839.805,E2 -18839.805} C_VEL
LIN {X 0,Y 264.997,Z 1011.722,A -85,B 0,C 180,E1 -18842.033,E2 -18842.033} C_VEL
LIN {X 0,Y 268.153,Z 1003.155,A -85,B 0,C 180,E1 -18843.843,E2 -18843.843} C_VEL
LIN {X 0,Y 271.865,Z 992.378,A -85,B 0,C 180,E1 -18845.793,E2 -18845.793} C_VEL
LIN {X 0,Y 275.737,Z 981.134,A -85,B 0,C 180,E1 -18847.482,E2 -18847.482} C_VEL
LIN {X 0,Y 279.282,Z 969.468,A -85,B 0,C 180,E1 -18848.984,E2 -18848.984} C_VEL
LIN {X 0,Y 282.587,Z 957.446,A -85,B 0,C 180,E1 -18850.286,E2 -18850.286} C_VEL
LIN {X 0,Y 285.665,Z 945.132,A -85,B 0,C 180,E1 -18851.389,E2 -18851.389} C_VEL
LIN {X 0,Y 288.303,Z 932.589,A -85,B 0,C 180,E1 -18852.33,E2 -18852.33} C_VEL
LIN {X 0,Y 290.788,Z 919.167,A -85,B 0,C 180,E1 -18853.118,E2 -18853.118} C_VEL
LIN {X 0,Y 292.774,Z 906.256,A -85,B 0,C 180,E1 -18853.699,E2 -18853.699} C_VEL
LIN {X 0,Y 294.242,Z 893.495,A -85,B 0,C 180,E1 -18854.134,E2 -18854.134} C_VEL
LIN {X 0,Y 295.799,Z 866.727,A -85,B 0,C 180,E1 -18854.819,E2 -18854.819} C_VEL
LIN {X 0,Y 301.061,Z 772.182,A -85,B 0,C 180,E1 -18856.975,E2 -18856.975} C_VEL
LIN {X 0,Y 300.326,Z 770.082,A -85,B 0,C 180,E1 -18857.196,E2 -18857.196} C_VEL
LIN {X 0,Y 293.938,Z 755.968,A -85,B 0,C 180,E1 -18859.059,E2 -18859.059} C_VEL
LIN {X 0,Y 286.907,Z 742.071,A -85,B 0,C 180,E1 -18861.232,E2 -18861.232} C_VEL
LIN {X 0,Y 279.591,Z 729.038,A -85,B 0,C 180,E1 -18863.672,E2 -18863.672} C_VEL
LIN {X 0,Y 272.901,Z 718.303,A -85,B 0,C 180,E1 -18866.103,E2 -18866.103} C_VEL
LIN {X 0,Y 268.754,Z 712.052,A -85,B 0,C 180,E1 -18867.735,E2 -18867.735} C_VEL
LIN {X 0,Y 266.019,Z 708.436,A -85,B 0,C 180,E1 -18868.856,E2 -18868.856} C_VEL
LIN {X 0,Y 263.098,Z 704.824,A -85,B 0,C 180,E1 -18870.109,E2 -18870.109} C_VEL
LIN {X 0,Y 262.139,Z 703.558,A -85,B 0,C 180,E1 -18870.541,E2 -18870.541} C_VEL
LIN {X 0,Y 259.411,Z 700.542,A -85,B 0,C 180,E1 -18871.788,E2 -18871.788} C_VEL
LIN {X 0,Y 258.148,Z 698.483,A -85,B 0,C 180,E1 -18872.431,E2 -18872.431} C_VEL
LIN {X 0,Y 255.584,Z 696.274,A -85,B 0,C 180,E1 -18873.679,E2 -18873.679} C_VEL
LIN {X 0,Y 253.709,Z 693.132,A -85,B 0,C 180,E1 -18874.742,E2 -18874.742} C_VEL
LIN {X 0,Y 250.666,Z 690.941,A -85,B 0,C 180,E1 -18876.396,E2 -18876.396} C_VEL
LIN {X 0,Y 249.273,Z 688.308,A -85,B 0,C 180,E1 -18877.409,E2 -18877.409} C_VEL
LIN {X 0,Y 249.074,Z 687.292,A -85,B 0,C 180,E1 -18878.209,E2 -18878.209} C_VEL
LIN {X 0,Y 249.13,Z 687.242,A -85,B 0,C 180,E1 -18881.922,E2 -18881.922} C_VEL
LIN {X 0,Y 249.191,Z 687.246,A -85,B 0,C 180,E1 -18885.295,E2 -18885.295} C_VEL
LIN {X 0,Y 249.419,Z 687.212,A -85,B 0,C 180,E1 -18890.465,E2 -18890.465} C_VEL
LIN {X 0,Y 249.454,Z 687.205,A -85,B 0,C 180,E1 -18893.529,E2 -18893.529} C_VEL
LIN {X 0,Y 249.67,Z 687.175,A -85,B 0,C 180,E1 -18898.387,E2 -18898.387} C_VEL
LIN {X 0,Y 249.67,Z 687.173,A -85,B 0,C 180,E1 -18901.613,E2 -18901.613} C_VEL
LIN {X 0,Y 249.443,Z 687.204,A -85,B 0,C 180,E1 -18906.725,E2 -18906.725} C_VEL
LIN {X 0,Y 249.383,Z 687.225,A -85,B 0,C 180,E1 -18909.734,E2 -18909.734} C_VEL
LIN {X 0,Y 249.194,Z 687.246,A -85,B 0,C 180,E1 -18914.704,E2 -18914.704} C_VEL
LIN {X 0,Y 249.142,Z 687.239,A -85,B 0,C 180,E1 -18918.077,E2 -18918.077} C_VEL
LIN {X 0,Y 249.094,Z 687.422,A -85,B 0,C 180,E1 -18922.388,E2 -18922.388} C_VEL
LIN {X 0,Y 249.367,Z 688.599,A -85,B 0,C 180,E1 -18923.128,E2 -18923.128} C_VEL
LIN {X 0,Y 250.795,Z 691.027,A -85,B 0,C 180,E1 -18924.084,E2 -18924.084} C_VEL
LIN {X 0,Y 253.989,Z 693.541,A -85,B 0,C 180,E1 -18925.824,E2 -18925.824} C_VEL
LIN {X 0,Y 255.895,Z 696.647,A -85,B 0,C 180,E1 -18926.891,E2 -18926.891} C_VEL
LIN {X 0,Y 258.527,Z 699.002,A -85,B 0,C 180,E1 -18928.166,E2 -18928.166} C_VEL
LIN {X 0,Y 260.823,Z 702.374,A -85,B 0,C 180,E1 -18929.289,E2 -18929.289} C_VEL
LIN {X 0,Y 262.875,Z 704.452,A -85,B 0,C 180,E1 -18930.195,E2 -18930.195} C_VEL
LIN {X 0,Y 265.66,Z 708.09,A -85,B 0,C 180,E1 -18931.406,E2 -18931.406} C_VEL
LIN {X 0,Y 267.257,Z 710.018,A -85,B 0,C 180,E1 -18932.063,E2 -18932.063} C_VEL
LIN {X 0,Y 271.254,Z 715.197,A -85,B 0,C 180,E1 -18933.641,E2 -18933.641} C_VEL
LIN {X 0,Y 274.342,Z 719.347,A -85,B 0,C 180,E1 -18934.794,E2 -18934.794} C_VEL
LIN {X 0,Y 285.217,Z 733.164,A -85,B 0,C 180,E1 -18938.4,E2 -18938.4} C_VEL
LIN {X 0,Y 292.208,Z 740.415,A -85,B 0,C 180,E1 -18940.381,E2 -18940.381} C_VEL
LIN {X 0,Y 298.506,Z 746.511,A -85,B 0,C 180,E1 -18942.144,E2 -18942.144} C_VEL
LIN {X 0,Y 302.07,Z 749.845,A -85,B 0,C 180,E1 -18943.196,E2 -18943.196} C_VEL
LIN {X 0,Y 306.974,Z 754.204,A -85,B 0,C 180,E1 -18944.696,E2 -18944.696} C_VEL
LIN {X 0,Y 312.985,Z 759.919,A -85,B 0,C 180,E1 -18946.686,E2 -18946.686} C_VEL
LIN {X 0,Y 319.507,Z 766.199,A -85,B 0,C 180,E1 -18949.077,E2 -18949.077} C_VEL
LIN {X 0,Y 322.961,Z 769.567,A -85,B 0,C 180,E1 -18950.405,E2 -18950.405} C_VEL
LIN {X 0,Y 327.584,Z 773.726,A -85,B 0,C 180,E1 -18952.224,E2 -18952.224} C_VEL
LIN {X 0,Y 333.059,Z 779.067,A -85,B 0,C 180,E1 -18954.471,E2 -18954.471} C_VEL
LIN {X 0,Y 336.557,Z 782.063,A -85,B 0,C 180,E1 -18955.945,E2 -18955.945} C_VEL
LIN {X 0,Y 341.268,Z 786.427,A -85,B 0,C 180,E1 -18958.033,E2 -18958.033} C_VEL
LIN {X 0,Y 344.244,Z 789.007,A -85,B 0,C 180,E1 -18959.392,E2 -18959.392} C_VEL
LIN {X 0,Y 348.426,Z 792.893,A -85,B 0,C 180,E1 -18961.394,E2 -18961.394} C_VEL
LIN {X 0,Y 351.624,Z 795.377,A -85,B 0,C 180,E1 -18962.995,E2 -18962.995} C_VEL
LIN {X 0,Y 354.988,Z 798.786,A -85,B 0,C 180,E1 -18964.814,E2 -18964.814} C_VEL
LIN {X 0,Y 359.263,Z 801.852,A -85,B 0,C 180,E1 -18967.22,E2 -18967.22} C_VEL
LIN {X 0,Y 360.657,Z 803.102,A -85,B 0,C 180,E1 -18968.055,E2 -18968.055} C_VEL
LIN {X 0,Y 364.005,Z 806.371,A -85,B 0,C 180,E1 -18970.277,E2 -18970.277} C_VEL
LIN {X 0,Y 367.434,Z 808.704,A -85,B 0,C 180,E1 -18972.698,E2 -18972.698} C_VEL
LIN {X 0,Y 369.169,Z 809.871,A -85,B 0,C 180,E1 -18974.053,E2 -18974.053} C_VEL
LIN {X 0,Y 371.65,Z 812.628,A -85,B 0,C 180,E1 -18976.341,E2 -18976.341} C_VEL
LIN {X 0,Y 373.779,Z 814.379,A -85,B 0,C 180,E1 -18978.539,E2 -18978.539} C_VEL
LIN {X 0,Y 375.614,Z 815.469,A -85,B 0,C 180,E1 -18980.831,E2 -18980.831} C_VEL
LIN {X 0,Y 377.362,Z 816.223,A -85,B 0,C 180,E1 -18983.584,E2 -18983.584} C_VEL
LIN {X 0,Y 378.239,Z 816.847,A -85,B 0,C 180,E1 -18985.738,E2 -18985.738} C_VEL
LIN {X 0,Y 378.813,Z 817.057,A -85,B 0,C 180,E1 -18987.874,E2 -18987.874} C_VEL
LIN {X 0,Y 379.014,Z 817.143,A -85,B 0,C 180,E1 -18990,E2 -18990} C_VEL
LIN {X 0,Y 378.813,Z 817.057,A -85,B 0,C 180,E1 -18992.126,E2 -18992.126} C_VEL
LIN {X 0,Y 378.094,Z 816.715,A -85,B 0,C 180,E1 -18994.715,E2 -18994.715} C_VEL
LIN {X 0,Y 376.835,Z 816.059,A -85,B 0,C 180,E1 -18997.319,E2 -18997.319} C_VEL
LIN {X 0,Y 375.218,Z 815.301,A -85,B 0,C 180,E1 -18999.705,E2 -18999.705} C_VEL
LIN {X 0,Y 373.019,Z 813.819,A -85,B 0,C 180,E1 -19002.253,E2 -19002.253} C_VEL
LIN {X 0,Y 370.555,Z 811.531,A -85,B 0,C 180,E1 -19004.702,E2 -19004.702} C_VEL
LIN {X 0,Y 368.326,Z 809.164,A -85,B 0,C 180,E1 -19006.631,E2 -19006.631} C_VEL
LIN {X 0,Y 365.305,Z 807.35,A -85,B 0,C 180,E1 -19008.835,E2 -19008.835} C_VEL
LIN {X 0,Y 361.681,Z 804.239,A -85,B 0,C 180,E1 -19011.263,E2 -19011.263} C_VEL
LIN {X 0,Y 359.513,Z 801.961,A -85,B 0,C 180,E1 -19012.638,E2 -19012.638} C_VEL
LIN {X 0,Y 355.557,Z 799.231,A -85,B 0,C 180,E1 -19014.881,E2 -19014.881} C_VEL
LIN {X 0,Y 351.581,Z 795.353,A -85,B 0,C 180,E1 -19017.028,E2 -19017.028} C_VEL
LIN {X 0,Y 346.682,Z 791.433,A -85,B 0,C 180,E1 -19019.44,E2 -19019.44} C_VEL
LIN {X 0,Y 342.405,Z 787.302,A -85,B 0,C 180,E1 -19021.466,E2 -19021.466} C_VEL
LIN {X 0,Y 337.562,Z 783.07,A -85,B 0,C 180,E1 -19023.614,E2 -19023.614} C_VEL
LIN {X 0,Y 334.432,Z 780.149,A -85,B 0,C 180,E1 -19024.959,E2 -19024.959} C_VEL
LIN {X 0,Y 329.365,Z 775.567,A -85,B 0,C 180,E1 -19027.048,E2 -19027.048} C_VEL
LIN {X 0,Y 326.433,Z 772.808,A -85,B 0,C 180,E1 -19028.23,E2 -19028.23} C_VEL
LIN {X 0,Y 321.626,Z 768.139,A -85,B 0,C 180,E1 -19030.112,E2 -19030.112} C_VEL
LIN {X 0,Y 315.791,Z 762.598,A -85,B 0,C 180,E1 -19032.32,E2 -19032.32} C_VEL
LIN {X 0,Y 308.821,Z 756.024,A -85,B 0,C 180,E1 -19034.714,E2 -19034.714} C_VEL
LIN {X 0,Y 302.28,Z 750.064,A -85,B 0,C 180,E1 -19036.736,E2 -19036.736} C_VEL
LIN {X 0,Y 299.01,Z 746.944,A -85,B 0,C 180,E1 -19037.717,E2 -19037.717} C_VEL
LIN {X 0,Y 293.404,Z 741.561,A -85,B 0,C 180,E1 -19039.289,E2 -19039.289} C_VEL
LIN {X 0,Y 287.064,Z 735.157,A -85,B 0,C 180,E1 -19041.056,E2 -19041.056} C_VEL
LIN {X 0,Y 281.038,Z 728.122,A -85,B 0,C 180,E1 -19042.906,E2 -19042.906} C_VEL
LIN {X 0,Y 271.734,Z 715.856,A -85,B 0,C 180,E1 -19046.175,E2 -19046.175} C_VEL
LIN {X 0,Y 269.218,Z 712.586,A -85,B 0,C 180,E1 -19047.147,E2 -19047.147} C_VEL
LIN {X 0,Y 266.023,Z 708.426,A -85,B 0,C 180,E1 -19048.448,E2 -19048.448} C_VEL
LIN {X 0,Y 263.25,Z 705.068,A -85,B 0,C 180,E1 -19049.631,E2 -19049.631} C_VEL
LIN {X 0,Y 262.101,Z 703.52,A -85,B 0,C 180,E1 -19050.15,E2 -19050.15} C_VEL
LIN {X 0,Y 259.41,Z 700.558,A -85,B 0,C 180,E1 -19051.38,E2 -19051.38} C_VEL
LIN {X 0,Y 258.27,Z 698.539,A -85,B 0,C 180,E1 -19051.969,E2 -19051.969} C_VEL
LIN {X 0,Y 255.638,Z 696.306,A -85,B 0,C 180,E1 -19053.245,E2 -19053.245} C_VEL
LIN {X 0,Y 253.549,Z 693.013,A -85,B 0,C 180,E1 -19054.418,E2 -19054.418} C_VEL
LIN {X 0,Y 250.796,Z 691.018,A -85,B 0,C 180,E1 -19055.916,E2 -19055.916} C_VEL
LIN {X 0,Y 249.297,Z 688.397,A -85,B 0,C 180,E1 -19056.974,E2 -19056.974} C_VEL
LIN {X 0,Y 249.09,Z 687.365,A -85,B 0,C 180,E1 -19057.72,E2 -19057.72} C_VEL
LIN {X 0,Y 249.142,Z 687.239,A -85,B 0,C 180,E1 -19061.923,E2 -19061.923} C_VEL
LIN {X 0,Y 249.194,Z 687.245,A -85,B 0,C 180,E1 -19065.296,E2 -19065.296} C_VEL
LIN {X 0,Y 249.418,Z 687.215,A -85,B 0,C 180,E1 -19070.466,E2 -19070.466} C_VEL
LIN {X 0,Y 249.453,Z 687.204,A -85,B 0,C 180,E1 -19073.53,E2 -19073.53} C_VEL
LIN {X 0,Y 249.67,Z 687.174,A -85,B 0,C 180,E1 -19078.387,E2 -19078.387} C_VEL
LIN {X 0,Y 249.67,Z 687.177,A -85,B 0,C 180,E1 -19081.613,E2 -19081.613} C_VEL
LIN {X 0,Y 249.454,Z 687.206,A -85,B 0,C 180,E1 -19086.471,E2 -19086.471} C_VEL
LIN {X 0,Y 249.383,Z 687.218,A -85,B 0,C 180,E1 -19089.735,E2 -19089.735} C_VEL
LIN {X 0,Y 249.191,Z 687.243,A -85,B 0,C 180,E1 -19094.705,E2 -19094.705} C_VEL
LIN {X 0,Y 249.13,Z 687.24,A -85,B 0,C 180,E1 -19098.078,E2 -19098.078} C_VEL
LIN {X 0,Y 249.094,Z 687.429,A -85,B 0,C 180,E1 -19101.953,E2 -19101.953} C_VEL
LIN {X 0,Y 249.396,Z 688.66,A -85,B 0,C 180,E1 -19102.743,E2 -19102.743} C_VEL
LIN {X 0,Y 250.744,Z 691.03,A -85,B 0,C 180,E1 -19103.651,E2 -19103.651} C_VEL
LIN {X 0,Y 253.984,Z 693.521,A -85,B 0,C 180,E1 -19105.413,E2 -19105.413} C_VEL
LIN {X 0,Y 255.671,Z 696.375,A -85,B 0,C 180,E1 -19106.367,E2 -19106.367} C_VEL
LIN {X 0,Y 258.479,Z 698.917,A -85,B 0,C 180,E1 -19107.734,E2 -19107.734} C_VEL
LIN {X 0,Y 260.934,Z 702.467,A -85,B 0,C 180,E1 -19108.931,E2 -19108.931} C_VEL
LIN {X 0,Y 262.817,Z 704.366,A -85,B 0,C 180,E1 -19109.761,E2 -19109.761} C_VEL
LIN {X 0,Y 265.634,Z 708.085,A -85,B 0,C 180,E1 -19110.99,E2 -19110.99} C_VEL
LIN {X 0,Y 267.268,Z 710.057,A -85,B 0,C 180,E1 -19111.662,E2 -19111.662} C_VEL
LIN {X 0,Y 271.321,Z 715.895,A -85,B 0,C 180,E1 -19113.289,E2 -19113.289} C_VEL
LIN {X 0,Y 274.935,Z 721.556,A -85,B 0,C 180,E1 -19114.664,E2 -19114.664} C_VEL
LIN {X 0,Y 280.918,Z 731.377,A -85,B 0,C 180,E1 -19116.79,E2 -19116.79} C_VEL
LIN {X 0,Y 287.608,Z 743.436,A -85,B 0,C 180,E1 -19118.993,E2 -19118.993} C_VEL
LIN {X 0,Y 294.915,Z 757.943,A -85,B 0,C 180,E1 -19121.229,E2 -19121.229} C_VEL
LIN {X 0,Y 295.175,Z 758.578,A -85,B 0,C 180,E1 -19121.309,E2 -19121.309} C_VEL
LIN {X 0,Y 296.227,Z 761.902,A -85,B 0,C 180,E1 -19121.657,E2 -19121.657} C_VEL
LIN {X 0,Y 296.909,Z 767.506,A -85,B 0,C 180,E1 -19122.001,E2 -19122.001} C_VEL
LIN {X 0,Y 296.813,Z 773.409,A -85,B 0,C 180,E1 -19122.189,E2 -19122.189} C_VEL
LIN {X 0,Y 295.264,Z 789.935,A -85,B 0,C 180,E1 -19122.443,E2 -19122.443} C_VEL
LIN {X 0,Y 289.411,Z 889.675,A -85,B 0,C 180,E1 -19124.768,E2 -19124.768} C_VEL
LIN {X 0,Y 288.198,Z 902.135,A -85,B 0,C 180,E1 -19125.179,E2 -19125.179} C_VEL
LIN {X 0,Y 286.319,Z 915.235,A -85,B 0,C 180,E1 -19125.732,E2 -19125.732} C_VEL
LIN {X 0,Y 284.019,Z 927.598,A -85,B 0,C 180,E1 -19126.39,E2 -19126.39} C_VEL
LIN {X 0,Y 281.722,Z 938.983,A -85,B 0,C 180,E1 -19127.174,E2 -19127.174} C_VEL
LIN {X 0,Y 278.536,Z 952.215,A -85,B 0,C 180,E1 -19128.281,E2 -19128.281} C_VEL
LIN {X 0,Y 275.441,Z 963.51,A -85,B 0,C 180,E1 -19129.411,E2 -19129.411} C_VEL
LIN {X 0,Y 271.638,Z 975.985,A -85,B 0,C 180,E1 -19130.912,E2 -19130.912} C_VEL
LIN {X 0,Y 268.094,Z 986.736,A -85,B 0,C 180,E1 -19132.449,E2 -19132.449} C_VEL
LIN {X 0,Y 264.285,Z 997.229,A -85,B 0,C 180,E1 -19134.196,E2 -19134.196} C_VEL
LIN {X 0,Y 260.84,Z 1006.497,A -85,B 0,C 180,E1 -19136.009,E2 -19136.009} C_VEL
LIN {X 0,Y 256.985,Z 1016.319,A -85,B 0,C 180,E1 -19138.264,E2 -19138.264} C_VEL
LIN {X 0,Y 253.554,Z 1024.75,A -85,B 0,C 180,E1 -19140.529,E2 -19140.529} C_VEL
LIN {X 0,Y 250.077,Z 1033.351,A -85,B 0,C 180,E1 -19143.279,E2 -19143.279} C_VEL
LIN {X 0,Y 247.506,Z 1039.859,A -85,B 0,C 180,E1 -19145.722,E2 -19145.722} C_VEL
LIN {X 0,Y 244.731,Z 1047.05,A -85,B 0,C 180,E1 -19148.964,E2 -19148.964} C_VEL
LIN {X 0,Y 243.077,Z 1051.705,A -85,B 0,C 180,E1 -19151.456,E2 -19151.456} C_VEL
LIN {X 0,Y 241.49,Z 1056.812,A -85,B 0,C 180,E1 -19154.816,E2 -19154.816} C_VEL
LIN {X 0,Y 240.393,Z 1060.817,A -85,B 0,C 180,E1 -19158.191,E2 -19158.191} C_VEL
LIN {X 0,Y 239.906,Z 1063.784,A -85,B 0,C 180,E1 -19161.578,E2 -19161.578} C_VEL
LIN {X 0,Y 239.781,Z 1064.975,A -85,B 0,C 180,E1 -19163.267,E2 -19163.267} C_VEL
LIN {X 0,Y 239.743,Z 1066.452,A -85,B 0,C 180,E1 -19166.639,E2 -19166.639} C_VEL
LIN {X 0,Y 239.89,Z 1066.946,A -85,B 0,C 180,E1 -19170,E2 -19170} C_VEL
LIN {X 0,Y 239.743,Z 1066.452,A -85,B 0,C 180,E1 -19173.361,E2 -19173.361} C_VEL
LIN {X 0,Y 239.781,Z 1064.975,A -85,B 0,C 180,E1 -19176.733,E2 -19176.733} C_VEL
LIN {X 0,Y 240.091,Z 1062.496,A -85,B 0,C 180,E1 -19180.115,E2 -19180.115} C_VEL
LIN {X 0,Y 241.174,Z 1057.902,A -85,B 0,C 180,E1 -19184.341,E2 -19184.341} C_VEL
LIN {X 0,Y 242.192,Z 1054.406,A -85,B 0,C 180,E1 -19186.868,E2 -19186.868} C_VEL
LIN {X 0,Y 244.129,Z 1048.673,A -85,B 0,C 180,E1 -19190.209,E2 -19190.209} C_VEL
LIN {X 0,Y 246.098,Z 1043.611,A -85,B 0,C 180,E1 -19192.676,E2 -19192.676} C_VEL
LIN {X 0,Y 248.736,Z 1036.685,A -85,B 0,C 180,E1 -19195.523,E2 -19195.523} C_VEL
LIN {X 0,Y 252.029,Z 1028.591,A -85,B 0,C 180,E1 -19198.297,E2 -19198.297} C_VEL
LIN {X 0,Y 255.34,Z 1020.626,A -85,B 0,C 180,E1 -19200.609,E2 -19200.609} C_VEL
LIN {X 0,Y 258.915,Z 1011.513,A -85,B 0,C 180,E1 -19202.879,E2 -19202.879} C_VEL
LIN {X 0,Y 262.222,Z 1002.948,A -85,B 0,C 180,E1 -19204.717,E2 -19204.717} C_VEL
LIN {X 0,Y 266.085,Z 992.171,A -85,B 0,C 180,E1 -19206.696,E2 -19206.696} C_VEL
LIN {X 0,Y 270.079,Z 980.926,A -85,B 0,C 180,E1 -19208.408,E2 -19208.408} C_VEL
LIN {X 0,Y 273.755,Z 969.261,A -85,B 0,C 180,E1 -19209.926,E2 -19209.926} C_VEL
LIN {X 0,Y 277.181,Z 957.239,A -85,B 0,C 180,E1 -19211.24,E2 -19211.24} C_VEL
LIN {X 0,Y 280.358,Z 944.926,A -85,B 0,C 180,E1 -19212.352,E2 -19212.352} C_VEL
LIN {X 0,Y 283.077,Z 932.383,A -85,B 0,C 180,E1 -19213.301,E2 -19213.301} C_VEL
LIN {X 0,Y 285.627,Z 918.961,A -85,B 0,C 180,E1 -19214.096,E2 -19214.096} C_VEL
LIN {X 0,Y 287.66,Z 906.049,A -85,B 0,C 180,E1 -19214.681,E2 -19214.681} C_VEL
LIN {X 0,Y 289.235,Z 892.554,A -85,B 0,C 180,E1 -19215.137,E2 -19215.137} C_VEL
LIN {X 0,Y 290.963,Z 863.61,A -85,B 0,C 180,E1 -19215.874,E2 -19215.874} C_VEL
LIN {X 0,Y 296.082,Z 774.296,A -85,B 0,C 180,E1 -19217.935,E2 -19217.935} C_VEL
LIN {X 0,Y 289.843,Z 760.219,A -85,B 0,C 180,E1 -19219.835,E2 -19219.835} C_VEL
LIN {X 0,Y 283.045,Z 746.627,A -85,B 0,C 180,E1 -19222.025,E2 -19222.025} C_VEL
LIN {X 0,Y 277.526,Z 736.574,A -85,B 0,C 180,E1 -19223.927,E2 -19223.927} C_VEL
LIN {X 0,Y 271.553,Z 726.477,A -85,B 0,C 180,E1 -19226.145,E2 -19226.145} C_VEL
LIN {X 0,Y 266.143,Z 718.085,A -85,B 0,C 180,E1 -19228.326,E2 -19228.326} C_VEL
LIN {X 0,Y 263.51,Z 714.562,A -85,B 0,C 180,E1 -19229.442,E2 -19229.442} C_VEL
LIN {X 0,Y 260.418,Z 710.532,A -85,B 0,C 180,E1 -19230.826,E2 -19230.826} C_VEL
LIN {X 0,Y 256.971,Z 706.482,A -85,B 0,C 180,E1 -19232.459,E2 -19232.459} C_VEL
LIN {X 0,Y 255.836,Z 704.818,A -85,B 0,C 180,E1 -19233.046,E2 -19233.046} C_VEL
LIN {X 0,Y 253.107,Z 702.08,A -85,B 0,C 180,E1 -19234.451,E2 -19234.451} C_VEL
LIN {X 0,Y 251.768,Z 699.718,A -85,B 0,C 180,E1 -19235.246,E2 -19235.246} C_VEL
LIN {X 0,Y 248.798,Z 697.391,A -85,B 0,C 180,E1 -19236.925,E2 -19236.925} C_VEL
LIN {X 0,Y 246.814,Z 694.048,A -85,B 0,C 180,E1 -19238.273,E2 -19238.273} C_VEL
LIN {X 0,Y 244.033,Z 692.204,A -85,B 0,C 180,E1 -19240.111,E2 -19240.111} C_VEL
LIN {X 0,Y 242.497,Z 689.848,A -85,B 0,C 180,E1 -19241.355,E2 -19241.355} C_VEL
LIN {X 0,Y 242.175,Z 688.628,A -85,B 0,C 180,E1 -19242.04,E2 -19242.04} C_VEL
LIN {X 0,Y 242.159,Z 688.136,A -85,B 0,C 180,E1 -19243.278,E2 -19243.278} C_VEL
LIN {X 0,Y 242.18,Z 688.111,A -85,B 0,C 180,E1 -19248.279,E2 -19248.279} C_VEL
LIN {X 0,Y 242.421,Z 688.072,A -85,B 0,C 180,E1 -19251.665,E2 -19251.665} C_VEL
LIN {X 0,Y 242.256,Z 688.114,A -85,B 0,C 180,E1 -19255.007,E2 -19255.007} C_VEL
LIN {X 0,Y 242.631,Z 688.051,A -85,B 0,C 180,E1 -19258.34,E2 -19258.34} C_VEL
LIN {X 0,Y 242.631,Z 688.049,A -85,B 0,C 180,E1 -19261.659,E2 -19261.659} C_VEL
LIN {X 0,Y 242.423,Z 688.078,A -85,B 0,C 180,E1 -19266.701,E2 -19266.701} C_VEL
LIN {X 0,Y 242.308,Z 688.111,A -85,B 0,C 180,E1 -19270.021,E2 -19270.021} C_VEL
